Yaskawa INFORM job: A_ROOF_SIDE_0617_2_PAINT_40.JBI

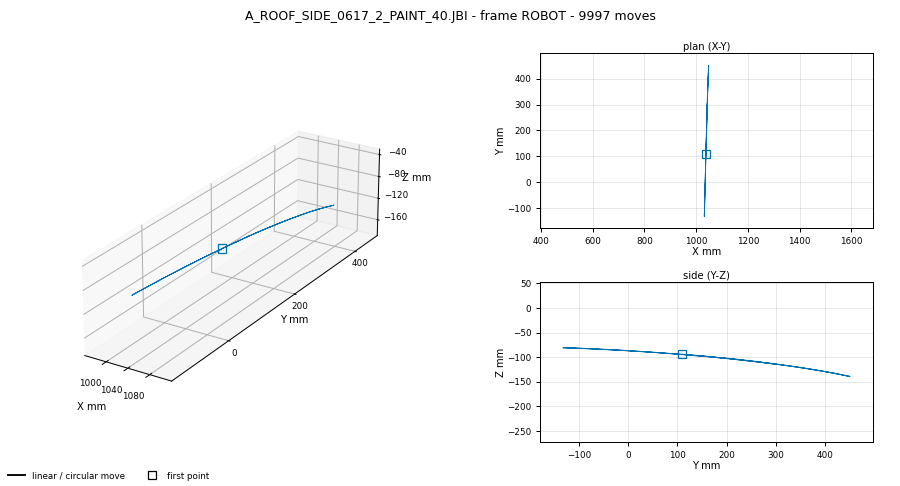
[picture p0: tool path of A_ROOF_SIDE_0617_2_PAINT_40.JBI in frame ROBOT, 9997 of 9997 moves have a stored position in this frame; points joined in program order, loops and branches not executed]
/JOB
//NAME A_ROOF_SIDE_0617_2_PAINT40
//POS
///NPOS 9997,0,0,0,0,0
///TOOL 1
///USER 0
///POSTYPE ROBOT
///RECTAN
///RCONF 1,0,0,0,0,0,0,0,0,0,0,0,0,0,0,0,0,0,0,0,0,0,0,0
C00000=1038.273,110.005,-93.623,169.688,40.047,157.538
C00001=1038.279,110.254,-93.643,169.691,40.048,157.539
C00002=1038.285,110.504,-93.663,169.693,40.048,157.539
C00003=1038.291,110.753,-93.683,169.696,40.048,157.539
C00004=1038.297,111.002,-93.703,169.698,40.048,157.539
C00005=1038.304,111.251,-93.723,169.700,40.048,157.539
C00006=1038.310,111.500,-93.743,169.702,40.049,157.539
C00007=1038.316,111.749,-93.762,169.704,40.049,157.539
C00008=1038.323,111.998,-93.782,169.706,40.049,157.539
C00009=1038.329,112.248,-93.802,169.708,40.050,157.540
C00010=1038.335,112.497,-93.822,169.710,40.049,157.540
C00011=1038.341,112.746,-93.842,169.713,40.050,157.540
C00012=1038.347,112.995,-93.862,169.715,40.050,157.540
C00013=1038.354,113.244,-93.882,169.717,40.050,157.540
C00014=1038.359,113.494,-93.903,169.719,40.051,157.540
C00015=1038.365,113.742,-93.923,169.721,40.051,157.540
C00016=1038.372,113.992,-93.943,169.723,40.051,157.540
C00017=1038.378,114.241,-93.963,169.725,40.051,157.541
C00018=1038.383,114.490,-93.984,169.727,40.052,157.541
C00019=1038.390,114.739,-94.004,169.730,40.052,157.541
C00020=1038.396,114.988,-94.024,169.732,40.052,157.541
C00021=1038.402,115.237,-94.044,169.734,40.052,157.541
C00022=1038.407,115.487,-94.065,169.736,40.053,157.541
C00023=1038.414,115.735,-94.085,169.738,40.053,157.542
C00024=1038.420,115.984,-94.105,169.740,40.053,157.542
C00025=1038.426,116.233,-94.126,169.742,40.054,157.542
C00026=1038.432,116.482,-94.146,169.745,40.054,157.542
C00027=1038.438,116.732,-94.167,169.747,40.054,157.542
C00028=1038.444,116.981,-94.187,169.749,40.054,157.542
C00029=1038.450,117.230,-94.207,169.751,40.055,157.542
C00030=1038.456,117.479,-94.227,169.753,40.055,157.543
C00031=1038.462,117.728,-94.247,169.755,40.056,157.543
C00032=1038.469,117.977,-94.268,169.757,40.055,157.543
C00033=1038.474,118.226,-94.289,169.759,40.056,157.543
C00034=1038.480,118.475,-94.309,169.762,40.056,157.543
C00035=1038.487,118.725,-94.329,169.765,40.057,157.543
C00036=1038.493,118.973,-94.349,169.767,40.057,157.543
C00037=1038.499,119.223,-94.370,169.769,40.057,157.544
C00038=1038.505,119.471,-94.391,169.771,40.057,157.544
C00039=1038.511,119.721,-94.411,169.773,40.058,157.544
C00040=1038.517,119.970,-94.431,169.775,40.058,157.544
C00041=1038.523,120.219,-94.452,169.777,40.058,157.544
C00042=1038.529,120.468,-94.472,169.780,40.059,157.544
C00043=1038.536,120.716,-94.493,169.782,40.059,157.544
C00044=1038.541,120.966,-94.514,169.784,40.059,157.544
C00045=1038.547,121.215,-94.534,169.786,40.059,157.545
C00046=1038.554,121.465,-94.554,169.788,40.060,157.545
C00047=1038.560,121.713,-94.575,169.790,40.060,157.545
C00048=1038.566,121.963,-94.596,169.792,40.060,157.545
C00049=1038.572,122.211,-94.615,169.794,40.060,157.545
C00050=1038.579,122.460,-94.637,169.797,40.061,157.545
C00051=1038.584,122.710,-94.657,169.800,40.061,157.545
C00052=1038.591,122.959,-94.677,169.802,40.061,157.546
C00053=1038.597,123.208,-94.697,169.804,40.062,157.546
C00054=1038.603,123.457,-94.719,169.806,40.061,157.546
C00055=1038.609,123.706,-94.739,169.808,40.062,157.546
C00056=1038.616,123.955,-94.759,169.810,40.062,157.546
C00057=1038.621,124.204,-94.781,169.812,40.063,157.546
C00058=1038.628,124.453,-94.801,169.814,40.062,157.546
C00059=1038.635,124.739,-94.825,169.818,40.063,157.547
C00060=1038.642,125.025,-94.849,169.820,40.063,157.547
C00061=1038.649,125.311,-94.871,169.822,40.064,157.547
C00062=1038.656,125.596,-94.895,169.825,40.064,157.547
C00063=1038.663,125.845,-94.916,169.827,40.064,157.547
C00064=1038.668,126.094,-94.937,169.829,40.064,157.547
C00065=1038.675,126.344,-94.957,169.831,40.065,157.548
C00066=1038.682,126.593,-94.978,169.833,40.065,157.548
C00067=1038.687,126.842,-94.999,169.836,40.065,157.548
C00068=1038.694,127.091,-95.020,169.838,40.065,157.548
C00069=1038.700,127.340,-95.040,169.840,40.065,157.548
C00070=1038.706,127.589,-95.061,169.843,40.066,157.548
C00071=1038.713,127.838,-95.082,169.845,40.066,157.548
C00072=1038.719,128.086,-95.102,169.847,40.067,157.549
C00073=1038.725,128.336,-95.123,169.849,40.066,157.549
C00074=1038.731,128.585,-95.143,169.851,40.067,157.549
C00075=1038.738,128.834,-95.164,169.854,40.067,157.549
C00076=1038.744,129.084,-95.185,169.856,40.067,157.549
C00077=1038.750,129.332,-95.206,169.858,40.068,157.549
C00078=1038.757,129.582,-95.226,169.861,40.068,157.549
C00079=1038.763,129.831,-95.248,169.863,40.068,157.549
C00080=1038.769,130.080,-95.268,169.865,40.068,157.550
C00081=1038.776,130.328,-95.289,169.867,40.069,157.550
C00082=1038.782,130.578,-95.310,169.869,40.068,157.550
C00083=1038.788,130.826,-95.330,169.872,40.069,157.550
C00084=1038.795,131.075,-95.351,169.874,40.069,157.550
C00085=1038.801,131.325,-95.372,169.877,40.070,157.550
C00086=1038.806,131.574,-95.394,169.879,40.070,157.551
C00087=1038.813,131.823,-95.415,169.881,40.070,157.551
C00088=1038.818,132.072,-95.435,169.883,40.070,157.551
C00089=1038.824,132.321,-95.457,169.885,40.071,157.551
C00090=1038.831,132.570,-95.478,169.888,40.071,157.551
C00091=1038.837,132.819,-95.498,169.890,40.072,157.551
C00092=1038.843,133.068,-95.520,169.892,40.072,157.551
C00093=1038.850,133.317,-95.541,169.894,40.073,157.552
C00094=1038.855,133.566,-95.562,169.896,40.072,157.552
C00095=1038.861,133.815,-95.583,169.899,40.073,157.552
C00096=1038.868,134.064,-95.604,169.901,40.073,157.552
C00097=1038.874,134.313,-95.626,169.904,40.074,157.552
C00098=1038.879,134.563,-95.646,169.906,40.074,157.552
C00099=1038.886,134.811,-95.668,169.908,40.075,157.553
C00100=1038.892,135.060,-95.689,169.910,40.074,157.553
C00101=1038.898,135.309,-95.710,169.912,40.075,157.553
C00102=1038.905,135.559,-95.731,169.914,40.075,157.553
C00103=1038.910,135.807,-95.752,169.917,40.076,157.553
C00104=1038.916,136.056,-95.774,169.920,40.076,157.553
C00105=1038.923,136.305,-95.795,169.922,40.076,157.554
C00106=1038.928,136.554,-95.815,169.924,40.076,157.554
C00107=1038.935,136.804,-95.837,169.926,40.077,157.554
C00108=1038.942,137.053,-95.858,169.928,40.077,157.554
C00109=1038.948,137.302,-95.880,169.930,40.078,157.554
C00110=1038.953,137.550,-95.901,169.933,40.078,157.554
C00111=1038.959,137.799,-95.922,169.936,40.078,157.554
C00112=1038.966,138.048,-95.944,169.938,40.079,157.555
C00113=1038.972,138.297,-95.964,169.940,40.079,157.555
C00114=1038.978,138.547,-95.986,169.942,40.079,157.555
C00115=1038.984,138.796,-96.007,169.944,40.080,157.555
C00116=1038.991,139.045,-96.028,169.947,40.080,157.555
C00117=1038.996,139.293,-96.050,169.949,40.080,157.555
C00118=1039.003,139.542,-96.071,169.952,40.081,157.556
C00119=1039.009,139.792,-96.093,169.954,40.081,157.556
C00120=1039.015,140.041,-96.115,169.956,40.082,157.556
C00121=1039.020,140.289,-96.136,169.958,40.082,157.556
C00122=1039.027,140.539,-96.157,169.960,40.083,157.556
C00123=1039.035,140.824,-96.182,169.963,40.083,157.556
C00124=1039.041,141.110,-96.206,169.966,40.083,157.557
C00125=1039.048,141.396,-96.232,169.969,40.084,157.557
C00126=1039.055,141.681,-96.255,169.971,40.084,157.557
C00127=1039.061,141.930,-96.277,169.973,40.085,157.557
C00128=1039.067,142.179,-96.299,169.976,40.085,157.557
C00129=1039.073,142.428,-96.320,169.978,40.085,157.558
C00130=1039.079,142.676,-96.342,169.981,40.086,157.558
C00131=1039.085,142.926,-96.364,169.983,40.086,157.558
C00132=1039.092,143.175,-96.386,169.985,40.087,157.558
C00133=1039.098,143.424,-96.407,169.987,40.087,157.558
C00134=1039.103,143.673,-96.429,169.990,40.088,157.558
C00135=1039.110,143.922,-96.450,169.992,40.088,157.559
C00136=1039.116,144.171,-96.472,169.995,40.088,157.559
C00137=1039.122,144.420,-96.493,169.997,40.089,157.559
C00138=1039.129,144.669,-96.514,169.999,40.089,157.559
C00139=1039.135,144.918,-96.536,170.001,40.089,157.559
C00140=1039.141,145.166,-96.558,170.004,40.089,157.559
C00141=1039.147,145.415,-96.580,170.006,40.090,157.560
C00142=1039.153,145.665,-96.601,170.008,40.090,157.560
C00143=1039.159,145.914,-96.623,170.011,40.091,157.560
C00144=1039.165,146.163,-96.645,170.013,40.091,157.560
C00145=1039.172,146.412,-96.667,170.016,40.092,157.560
C00146=1039.178,146.661,-96.689,170.018,40.092,157.560
C00147=1039.184,146.909,-96.710,170.020,40.092,157.561
C00148=1039.190,147.159,-96.732,170.022,40.093,157.561
C00149=1039.196,147.408,-96.753,170.025,40.093,157.561
C00150=1039.202,147.656,-96.775,170.028,40.094,157.561
C00151=1039.209,147.906,-96.797,170.030,40.094,157.561
C00152=1039.215,148.155,-96.819,170.032,40.095,157.562
C00153=1039.220,148.404,-96.842,170.034,40.095,157.562
C00154=1039.226,148.652,-96.863,170.036,40.095,157.562
C00155=1039.232,148.901,-96.885,170.040,40.096,157.562
C00156=1039.238,149.151,-96.906,170.042,40.096,157.562
C00157=1039.245,149.399,-96.929,170.044,40.097,157.562
C00158=1039.251,149.648,-96.950,170.046,40.097,157.563
C00159=1039.257,149.898,-96.972,170.048,40.098,157.563
C00160=1039.263,150.146,-96.995,170.051,40.098,157.563
C00161=1039.269,150.396,-97.016,170.054,40.099,157.563
C00162=1039.276,150.644,-97.039,170.056,40.099,157.563
C00163=1039.282,150.893,-97.060,170.058,40.100,157.564
C00164=1039.287,151.142,-97.082,170.060,40.100,157.564
C00165=1039.293,151.391,-97.105,170.063,40.101,157.564
C00166=1039.299,151.640,-97.126,170.066,40.101,157.564
C00167=1039.306,151.889,-97.149,170.068,40.102,157.564
C00168=1039.312,152.138,-97.170,170.070,40.102,157.565
C00169=1039.318,152.386,-97.193,170.073,40.102,157.565
C00170=1039.324,152.636,-97.215,170.075,40.103,157.565
C00171=1039.330,152.885,-97.237,170.077,40.103,157.565
C00172=1039.336,153.134,-97.259,170.079,40.104,157.565
C00173=1039.343,153.382,-97.281,170.083,40.104,157.565
C00174=1039.349,153.632,-97.303,170.085,40.104,157.566
C00175=1039.355,153.880,-97.326,170.087,40.105,157.566
C00176=1039.361,154.130,-97.347,170.089,40.106,157.566
C00177=1039.367,154.378,-97.370,170.091,40.106,157.566
C00178=1039.373,154.627,-97.391,170.095,40.107,157.567
C00179=1039.379,154.876,-97.414,170.097,40.107,157.567
C00180=1039.385,155.126,-97.436,170.099,40.108,157.567
C00181=1039.391,155.374,-97.459,170.101,40.108,157.567
C00182=1039.397,155.624,-97.481,170.104,40.108,157.567
C00183=1039.404,155.872,-97.503,170.107,40.109,157.568
C00184=1039.409,156.121,-97.526,170.109,40.110,157.568
C00185=1039.416,156.370,-97.547,170.111,40.110,157.568
C00186=1039.422,156.619,-97.570,170.114,40.111,157.568
C00187=1039.429,156.904,-97.595,170.116,40.111,157.568
C00188=1039.435,157.189,-97.621,170.120,40.112,157.569
C00189=1039.442,157.475,-97.646,170.122,40.113,157.569
C00190=1039.449,157.760,-97.672,170.125,40.113,157.569
C00191=1039.456,158.009,-97.694,170.127,40.113,157.569
C00192=1039.462,158.257,-97.716,170.130,40.114,157.569
C00193=1039.468,158.506,-97.739,170.133,40.115,157.570
C00194=1039.474,158.755,-97.762,170.135,40.115,157.570
C00195=1039.480,159.004,-97.784,170.137,40.116,157.570
C00196=1039.486,159.253,-97.806,170.140,40.116,157.570
C00197=1039.493,159.502,-97.829,170.142,40.116,157.570
C00198=1039.498,159.751,-97.852,170.144,40.117,157.571
C00199=1039.505,160.000,-97.874,170.147,40.118,157.571
C00200=1039.511,160.249,-97.897,170.150,40.118,157.571
C00201=1039.517,160.498,-97.919,170.152,40.119,157.571
C00202=1039.523,160.747,-97.942,170.154,40.120,157.572
C00203=1039.529,160.996,-97.965,170.157,40.120,157.572
C00204=1039.535,161.245,-97.988,170.160,40.121,157.572
C00205=1039.540,161.494,-98.010,170.162,40.122,157.572
C00206=1039.546,161.743,-98.032,170.164,40.122,157.572
C00207=1039.552,161.992,-98.055,170.166,40.122,157.573
C00208=1039.558,162.241,-98.078,170.170,40.123,157.573
C00209=1039.564,162.489,-98.101,170.172,40.124,157.573
C00210=1039.570,162.738,-98.124,170.174,40.124,157.573
C00211=1039.576,162.987,-98.146,170.176,40.125,157.574
C00212=1039.582,163.236,-98.169,170.179,40.126,157.574
C00213=1039.587,163.485,-98.192,170.182,40.127,157.574
C00214=1039.593,163.734,-98.215,170.184,40.127,157.574
C00215=1039.599,163.982,-98.238,170.187,40.128,157.574
C00216=1039.605,164.231,-98.261,170.189,40.129,157.575
C00217=1039.611,164.480,-98.284,170.192,40.129,157.575
C00218=1039.617,164.729,-98.306,170.194,40.130,157.575
C00219=1039.623,164.978,-98.330,170.197,40.131,157.575
C00220=1039.629,165.227,-98.352,170.199,40.131,157.576
C00221=1039.635,165.476,-98.375,170.202,40.132,157.576
C00222=1039.641,165.725,-98.398,170.204,40.132,157.576
C00223=1039.647,165.974,-98.421,170.207,40.133,157.576
C00224=1039.652,166.223,-98.444,170.209,40.134,157.577
C00225=1039.659,166.471,-98.467,170.211,40.134,157.577
C00226=1039.665,166.719,-98.490,170.215,40.135,157.577
C00227=1039.671,166.969,-98.513,170.217,40.136,157.577
C00228=1039.677,167.218,-98.536,170.219,40.136,157.577
C00229=1039.683,167.467,-98.559,170.222,40.137,157.578
C00230=1039.689,167.715,-98.582,170.224,40.138,157.578
C00231=1039.695,167.964,-98.604,170.227,40.139,157.578
C00232=1039.701,168.213,-98.627,170.230,40.139,157.579
C00233=1039.707,168.462,-98.651,170.232,40.139,157.579
C00234=1039.713,168.711,-98.674,170.234,40.140,157.579
C00235=1039.719,168.960,-98.697,170.238,40.141,157.579
C00236=1039.725,169.209,-98.720,170.240,40.142,157.579
C00237=1039.731,169.458,-98.743,170.242,40.142,157.580
C00238=1039.737,169.706,-98.766,170.245,40.143,157.580
C00239=1039.743,169.955,-98.790,170.248,40.144,157.580
C00240=1039.749,170.204,-98.813,170.250,40.144,157.580
C00241=1039.756,170.453,-98.835,170.253,40.145,157.581
C00242=1039.761,170.702,-98.858,170.255,40.146,157.581
C00243=1039.768,170.951,-98.882,170.257,40.146,157.581
C00244=1039.774,171.200,-98.905,170.261,40.147,157.581
C00245=1039.779,171.449,-98.928,170.263,40.147,157.582
C00246=1039.785,171.697,-98.951,170.265,40.148,157.582
C00247=1039.792,171.946,-98.975,170.268,40.149,157.582
C00248=1039.798,172.195,-98.997,170.271,40.149,157.582
C00249=1039.804,172.444,-99.020,170.273,40.150,157.583
C00250=1039.810,172.692,-99.044,170.276,40.151,157.583
C00251=1039.817,172.978,-99.070,170.279,40.152,157.583
C00252=1039.824,173.262,-99.097,170.282,40.152,157.583
C00253=1039.831,173.547,-99.123,170.285,40.153,157.584
C00254=1039.838,173.831,-99.150,170.288,40.154,157.584
C00255=1039.844,174.080,-99.173,170.290,40.154,157.584
C00256=1039.850,174.330,-99.196,170.294,40.155,157.584
C00257=1039.857,174.578,-99.220,170.296,40.156,157.585
C00258=1039.862,174.827,-99.243,170.298,40.156,157.585
C00259=1039.869,175.076,-99.267,170.301,40.157,157.585
C00260=1039.875,175.325,-99.289,170.303,40.158,157.585
C00261=1039.881,175.574,-99.312,170.307,40.159,157.586
C00262=1039.888,175.823,-99.336,170.309,40.159,157.586
C00263=1039.893,176.071,-99.359,170.311,40.160,157.586
C00264=1039.899,176.320,-99.383,170.314,40.160,157.586
C00265=1039.906,176.569,-99.406,170.317,40.161,157.587
C00266=1039.912,176.818,-99.430,170.320,40.162,157.587
C00267=1039.918,177.067,-99.453,170.322,40.162,157.587
C00268=1039.925,177.315,-99.476,170.324,40.163,157.587
C00269=1039.931,177.564,-99.499,170.328,40.164,157.587
C00270=1039.937,177.813,-99.523,170.330,40.165,157.588
C00271=1039.943,178.062,-99.546,170.333,40.165,157.588
C00272=1039.949,178.310,-99.570,170.335,40.166,157.588
C00273=1039.955,178.560,-99.593,170.339,40.166,157.589
C00274=1039.961,178.808,-99.617,170.341,40.168,157.589
C00275=1039.968,179.058,-99.640,170.344,40.168,157.589
C00276=1039.974,179.306,-99.664,170.346,40.169,157.589
C00277=1039.981,179.555,-99.687,170.350,40.169,157.590
C00278=1039.987,179.804,-99.710,170.352,40.170,157.590
C00279=1039.994,180.053,-99.734,170.354,40.171,157.590
C00280=1039.999,180.301,-99.757,170.357,40.171,157.590
C00281=1040.005,180.550,-99.781,170.359,40.172,157.591
C00282=1040.012,180.799,-99.805,170.363,40.172,157.591
C00283=1040.018,181.048,-99.828,170.365,40.174,157.591
C00284=1040.024,181.297,-99.852,170.368,40.174,157.591
C00285=1040.030,181.545,-99.876,170.370,40.175,157.592
C00286=1040.037,181.794,-99.899,170.374,40.175,157.592
C00287=1040.044,182.042,-99.922,170.376,40.176,157.592
C00288=1040.050,182.291,-99.946,170.379,40.177,157.592
C00289=1040.056,182.540,-99.969,170.381,40.178,157.593
C00290=1040.063,182.789,-99.993,170.385,40.178,157.593
C00291=1040.069,183.038,-100.017,170.387,40.179,157.593
C00292=1040.075,183.287,-100.041,170.390,40.179,157.593
C00293=1040.082,183.536,-100.064,170.392,40.180,157.594
C00294=1040.087,183.785,-100.088,170.396,40.181,157.594
C00295=1040.093,184.034,-100.112,170.398,40.182,157.594
C00296=1040.099,184.282,-100.136,170.401,40.183,157.594
C00297=1040.105,184.531,-100.160,170.404,40.184,157.595
C00298=1040.111,184.780,-100.184,170.406,40.185,157.595
C00299=1040.117,185.028,-100.208,170.409,40.186,157.595
C00300=1040.123,185.277,-100.232,170.411,40.186,157.596
C00301=1040.129,185.526,-100.257,170.415,40.187,157.596
C00302=1040.135,185.775,-100.281,170.417,40.188,157.596
C00303=1040.141,186.023,-100.305,170.420,40.189,157.597
C00304=1040.147,186.272,-100.329,170.423,40.190,157.597
C00305=1040.153,186.521,-100.353,170.426,40.191,157.597
C00306=1040.159,186.770,-100.377,170.428,40.192,157.597
C00307=1040.164,187.018,-100.402,170.431,40.193,157.598
C00308=1040.171,187.267,-100.426,170.434,40.194,157.598
C00309=1040.176,187.516,-100.450,170.437,40.195,157.598
C00310=1040.183,187.765,-100.474,170.439,40.196,157.599
C00311=1040.188,188.014,-100.498,170.443,40.196,157.599
C00312=1040.195,188.262,-100.522,170.445,40.197,157.599
C00313=1040.200,188.511,-100.546,170.448,40.198,157.599
C00314=1040.207,188.760,-100.570,170.450,40.199,157.600
C00315=1040.214,189.044,-100.598,170.454,40.200,157.600
C00316=1040.221,189.328,-100.625,170.457,40.201,157.600
C00317=1040.227,189.613,-100.654,170.460,40.202,157.601
C00318=1040.234,189.897,-100.681,170.463,40.203,157.601
C00319=1040.240,190.146,-100.705,170.466,40.204,157.601
C00320=1040.247,190.395,-100.730,170.469,40.205,157.602
C00321=1040.253,190.643,-100.754,170.472,40.206,157.602
C00322=1040.259,190.892,-100.779,170.475,40.207,157.602
C00323=1040.265,191.141,-100.802,170.477,40.208,157.603
C00324=1040.271,191.390,-100.827,170.481,40.209,157.603
C00325=1040.277,191.638,-100.852,170.483,40.209,157.603
C00326=1040.283,191.887,-100.876,170.486,40.210,157.604
C00327=1040.289,192.136,-100.900,170.488,40.211,157.604
C00328=1040.295,192.385,-100.925,170.492,40.212,157.604
C00329=1040.302,192.633,-100.949,170.494,40.213,157.605
C00330=1040.308,192.882,-100.974,170.497,40.214,157.605
C00331=1040.313,193.131,-100.998,170.500,40.215,157.605
C00332=1040.319,193.380,-101.022,170.503,40.216,157.606
C00333=1040.326,193.628,-101.047,170.506,40.217,157.606
C00334=1040.332,193.877,-101.071,170.509,40.218,157.606
C00335=1040.338,194.126,-101.096,170.512,40.219,157.606
C00336=1040.345,194.374,-101.120,170.514,40.220,157.607
C00337=1040.350,194.623,-101.145,170.518,40.221,157.607
C00338=1040.357,194.872,-101.169,170.520,40.222,157.607
C00339=1040.363,195.120,-101.194,170.523,40.223,157.608
C00340=1040.369,195.369,-101.218,170.527,40.224,157.608
C00341=1040.375,195.617,-101.243,170.529,40.225,157.608
C00342=1040.381,195.867,-101.268,170.532,40.226,157.609
C00343=1040.387,196.116,-101.292,170.534,40.227,157.609
C00344=1040.394,196.364,-101.317,170.538,40.228,157.609
C00345=1040.400,196.613,-101.341,170.541,40.229,157.610
C00346=1040.406,196.861,-101.366,170.543,40.230,157.610
C00347=1040.413,197.110,-101.390,170.547,40.231,157.610
C00348=1040.419,197.359,-101.415,170.549,40.232,157.611
C00349=1040.425,197.608,-101.439,170.552,40.233,157.611
C00350=1040.431,197.856,-101.464,170.556,40.233,157.611
C00351=1040.437,198.105,-101.489,170.558,40.234,157.611
C00352=1040.444,198.353,-101.514,170.561,40.235,157.612
C00353=1040.450,198.603,-101.538,170.565,40.236,157.612
C00354=1040.457,198.851,-101.563,170.567,40.237,157.612
C00355=1040.462,199.100,-101.587,170.570,40.238,157.613
C00356=1040.469,199.348,-101.612,170.572,40.239,157.613
C00357=1040.475,199.597,-101.637,170.576,40.240,157.613
C00358=1040.481,199.846,-101.662,170.579,40.241,157.614
C00359=1040.488,200.095,-101.686,170.581,40.242,157.614
C00360=1040.494,200.344,-101.711,170.585,40.243,157.614
C00361=1040.500,200.591,-101.736,170.588,40.244,157.615
C00362=1040.506,200.841,-101.760,170.590,40.245,157.615
C00363=1040.512,201.089,-101.786,170.594,40.246,157.615
C00364=1040.519,201.338,-101.811,170.597,40.247,157.616
C00365=1040.525,201.587,-101.835,170.600,40.248,157.616
C00366=1040.531,201.836,-101.860,170.603,40.249,157.616
C00367=1040.537,202.084,-101.885,170.606,40.250,157.617
C00368=1040.543,202.333,-101.910,170.609,40.251,157.617
C00369=1040.549,202.582,-101.935,170.612,40.253,157.618
C00370=1040.555,202.830,-101.961,170.614,40.254,157.618
C00371=1040.562,203.079,-101.986,170.618,40.255,157.618
C00372=1040.568,203.328,-102.011,170.621,40.256,157.619
C00373=1040.574,203.577,-102.036,170.623,40.257,157.619
C00374=1040.579,203.825,-102.061,170.627,40.259,157.619
C00375=1040.585,204.073,-102.086,170.630,40.259,157.620
C00376=1040.592,204.322,-102.112,170.632,40.261,157.620
C00377=1040.599,204.571,-102.136,170.636,40.261,157.620
C00378=1040.605,204.819,-102.162,170.639,40.263,157.621
C00379=1040.631,205.871,-102.268,170.925,40.366,157.654
C00380=1040.639,206.173,-102.300,170.927,40.368,157.655
C00381=1040.647,206.477,-102.333,170.930,40.370,157.656
C00382=1040.655,206.780,-102.365,170.933,40.373,157.656
C00383=1040.664,207.084,-102.396,170.935,40.375,157.657
C00384=1040.670,207.333,-102.423,170.938,40.377,157.657
C00385=1040.677,207.581,-102.449,170.939,40.379,157.658
C00386=1040.684,207.830,-102.476,170.942,40.380,157.658
C00387=1040.689,208.078,-102.502,170.944,40.383,157.659
C00388=1040.697,208.326,-102.530,170.946,40.384,157.659
C00389=1040.703,208.574,-102.556,170.948,40.386,157.660
C00390=1040.710,208.823,-102.583,170.951,40.388,157.660
C00391=1040.717,209.072,-102.609,170.952,40.390,157.661
C00392=1040.723,209.320,-102.635,170.955,40.392,157.661
C00393=1040.730,209.569,-102.662,170.957,40.393,157.662
C00394=1040.736,209.817,-102.688,170.959,40.396,157.662
C00395=1040.743,210.066,-102.715,170.962,40.397,157.663
C00396=1040.750,210.315,-102.742,170.964,40.399,157.663
C00397=1040.757,210.562,-102.768,170.967,40.401,157.664
C00398=1040.764,210.811,-102.795,170.968,40.403,157.664
C00399=1040.769,211.059,-102.821,170.971,40.405,157.665
C00400=1040.777,211.308,-102.848,170.973,40.407,157.665
C00401=1040.783,211.557,-102.875,170.976,40.409,157.666
C00402=1040.790,211.805,-102.902,170.977,40.410,157.666
C00403=1040.796,212.054,-102.929,170.980,40.413,157.667
C00404=1040.803,212.302,-102.955,170.982,40.414,157.667
C00405=1040.809,212.551,-102.982,170.984,40.416,157.668
C00406=1040.816,212.799,-103.009,170.986,40.418,157.668
C00407=1040.822,213.047,-103.035,170.989,40.420,157.669
C00408=1040.829,213.296,-103.062,170.991,40.422,157.669
C00409=1040.836,213.544,-103.090,170.993,40.424,157.670
C00410=1040.843,213.792,-103.116,170.995,40.426,157.670
C00411=1040.849,214.042,-103.143,170.998,40.428,157.671
C00412=1040.856,214.290,-103.170,171.001,40.430,157.671
C00413=1040.862,214.538,-103.196,171.002,40.431,157.672
C00414=1040.868,214.787,-103.223,171.005,40.434,157.672
C00415=1040.876,215.035,-103.251,171.007,40.435,157.673
C00416=1040.882,215.284,-103.277,171.010,40.437,157.673
C00417=1040.889,215.532,-103.304,171.012,40.439,157.674
C00418=1040.895,215.781,-103.331,171.014,40.441,157.674
C00419=1040.903,216.030,-103.358,171.016,40.443,157.675
C00420=1040.909,216.277,-103.385,171.019,40.444,157.675
C00421=1040.915,216.526,-103.412,171.021,40.446,157.676
C00422=1040.922,216.775,-103.439,171.023,40.448,157.676
C00423=1040.928,217.023,-103.466,171.025,40.450,157.676
C00424=1040.935,217.272,-103.492,171.028,40.452,157.677
C00425=1040.942,217.520,-103.520,171.030,40.454,157.678
C00426=1040.949,217.769,-103.547,171.033,40.455,157.678
C00427=1040.955,218.017,-103.574,171.035,40.458,157.679
C00428=1040.962,218.266,-103.601,171.037,40.459,157.679
C00429=1040.969,218.514,-103.628,171.040,40.461,157.679
C00430=1040.975,218.763,-103.655,171.042,40.463,157.680
C00431=1040.982,219.010,-103.682,171.045,40.465,157.681
C00432=1040.989,219.259,-103.709,171.047,40.467,157.681
C00433=1040.996,219.507,-103.736,171.049,40.468,157.681
C00434=1041.002,219.756,-103.763,171.051,40.471,157.682
C00435=1041.009,220.005,-103.791,171.054,40.472,157.682
C00436=1041.018,220.313,-103.824,171.056,40.474,157.683
C00437=1041.025,220.622,-103.858,171.060,40.477,157.684
C00438=1041.033,220.931,-103.892,171.063,40.479,157.684
C00439=1041.042,221.240,-103.926,171.065,40.482,157.685
C00440=1041.049,221.488,-103.954,171.068,40.483,157.685
C00441=1041.055,221.737,-103.981,171.071,40.486,157.686
C00442=1041.061,221.985,-104.008,171.073,40.487,157.687
C00443=1041.068,222.233,-104.036,171.076,40.489,157.687
C00444=1041.075,222.482,-104.062,171.077,40.491,157.688
C00445=1041.081,222.730,-104.090,171.080,40.493,157.688
C00446=1041.088,222.979,-104.118,171.082,40.495,157.688
C00447=1041.094,223.227,-104.145,171.085,40.497,157.689
C00448=1041.101,223.476,-104.172,171.087,40.498,157.690
C00449=1041.107,223.724,-104.200,171.090,40.500,157.690
C00450=1041.114,223.973,-104.227,171.092,40.502,157.691
C00451=1041.121,224.221,-104.255,171.094,40.504,157.691
C00452=1041.128,224.470,-104.282,171.097,40.506,157.692
C00453=1041.134,224.718,-104.309,171.099,40.508,157.692
C00454=1041.141,224.966,-104.337,171.101,40.510,157.693
C00455=1041.147,225.214,-104.364,171.104,40.512,157.693
C00456=1041.154,225.463,-104.392,171.107,40.513,157.694
C00457=1041.161,225.711,-104.420,171.109,40.515,157.694
C00458=1041.168,225.960,-104.446,171.112,40.517,157.695
C00459=1041.174,226.209,-104.474,171.114,40.519,157.695
C00460=1041.180,226.456,-104.501,171.116,40.521,157.696
C00461=1041.187,226.705,-104.529,171.118,40.523,157.696
C00462=1041.194,226.953,-104.557,171.121,40.525,157.697
C00463=1041.200,227.202,-104.585,171.123,40.526,157.697
C00464=1041.207,227.450,-104.612,171.126,40.529,157.698
C00465=1041.214,227.698,-104.640,171.128,40.530,157.698
C00466=1041.221,227.947,-104.668,171.131,40.532,157.699
C00467=1041.228,228.196,-104.694,171.134,40.534,157.699
C00468=1041.234,228.444,-104.722,171.136,40.536,157.700
C00469=1041.241,228.693,-104.750,171.139,40.537,157.700
C00470=1041.248,228.941,-104.777,171.141,40.540,157.701
C00471=1041.254,229.190,-104.806,171.144,40.541,157.701
C00472=1041.260,229.437,-104.834,171.146,40.543,157.702
C00473=1041.267,229.685,-104.862,171.149,40.545,157.702
C00474=1041.273,229.934,-104.889,171.150,40.547,157.703
C00475=1041.280,230.182,-104.917,171.153,40.549,157.703
C00476=1041.287,230.431,-104.945,171.155,40.551,157.704
C00477=1041.293,230.679,-104.972,171.158,40.553,157.704
C00478=1041.300,230.927,-105.000,171.161,40.555,157.705
C00479=1041.307,231.176,-105.028,171.163,40.556,157.705
C00480=1041.313,231.424,-105.056,171.166,40.558,157.706
C00481=1041.319,231.673,-105.084,171.168,40.560,157.706
C00482=1041.326,231.921,-105.112,171.171,40.562,157.707
C00483=1041.333,232.169,-105.140,171.173,40.564,157.707
C00484=1041.340,232.418,-105.168,171.176,40.566,157.708
C00485=1041.346,232.666,-105.196,171.179,40.568,157.708
C00486=1041.352,232.915,-105.224,171.181,40.569,157.709
C00487=1041.359,233.163,-105.252,171.184,40.572,157.709
C00488=1041.366,233.411,-105.280,171.186,40.573,157.710
C00489=1041.373,233.660,-105.308,171.189,40.576,157.710
C00490=1041.379,233.908,-105.336,171.191,40.577,157.711
C00491=1041.386,234.156,-105.365,171.194,40.579,157.712
C00492=1041.393,234.457,-105.398,171.197,40.582,157.712
C00493=1041.401,234.759,-105.432,171.200,40.584,157.713
C00494=1041.410,235.060,-105.466,171.203,40.586,157.713
C00495=1041.418,235.362,-105.501,171.206,40.588,157.714
C00496=1041.424,235.610,-105.529,171.208,40.590,157.715
C00497=1041.431,235.858,-105.556,171.211,40.592,157.715
C00498=1041.437,236.107,-105.585,171.213,40.594,157.715
C00499=1041.444,236.355,-105.613,171.217,40.596,157.716
C00500=1041.451,236.603,-105.641,171.219,40.597,157.717
C00501=1041.457,236.852,-105.670,171.222,40.600,157.717
C00502=1041.464,237.100,-105.698,171.224,40.601,157.718
C00503=1041.471,237.348,-105.726,171.227,40.604,157.718
C00504=1041.477,237.596,-105.754,171.230,40.605,157.719
C00505=1041.483,237.845,-105.782,171.232,40.607,157.719
C00506=1041.490,238.093,-105.811,171.235,40.609,157.720
C00507=1041.497,238.342,-105.839,171.237,40.611,157.720
C00508=1041.504,238.590,-105.868,171.240,40.613,157.721
C00509=1041.510,238.839,-105.895,171.242,40.615,157.721
C00510=1041.517,239.086,-105.924,171.245,40.617,157.722
C00511=1041.523,239.335,-105.952,171.248,40.618,157.722
C00512=1041.530,239.583,-105.981,171.250,40.620,157.723
C00513=1041.537,239.831,-106.008,171.253,40.622,157.723
C00514=1041.543,240.080,-106.037,171.255,40.624,157.724
C00515=1041.550,240.328,-106.065,171.258,40.626,157.724
C00516=1041.557,240.577,-106.094,171.260,40.628,157.725
C00517=1041.563,240.825,-106.122,171.263,40.630,157.726
C00518=1041.570,241.073,-106.151,171.267,40.631,157.726
C00519=1041.577,241.321,-106.180,171.269,40.634,157.727
C00520=1041.583,241.570,-106.207,171.272,40.635,157.727
C00521=1041.590,241.818,-106.237,171.274,40.638,157.728
C00522=1041.596,242.066,-106.266,171.277,40.639,157.728
C00523=1041.603,242.315,-106.294,171.279,40.641,157.729
C00524=1041.609,242.563,-106.323,171.282,40.643,157.729
C00525=1041.616,242.811,-106.351,171.285,40.645,157.730
C00526=1041.623,243.059,-106.380,171.287,40.647,157.730
C00527=1041.629,243.308,-106.408,171.290,40.649,157.731
C00528=1041.636,243.556,-106.437,171.292,40.651,157.731
C00529=1041.642,243.804,-106.466,171.295,40.653,157.732
C00530=1041.649,244.052,-106.495,171.297,40.655,157.732
C00531=1041.655,244.301,-106.523,171.301,40.657,157.733
C00532=1041.662,244.549,-106.552,171.304,40.658,157.733
C00533=1041.669,244.797,-106.581,171.306,40.660,157.734
C00534=1041.675,245.045,-106.610,171.309,40.662,157.735
C00535=1041.682,245.294,-106.638,171.311,40.664,157.735
C00536=1041.688,245.543,-106.667,171.314,40.667,157.736
C00537=1041.695,245.791,-106.696,171.317,40.668,157.736
C00538=1041.701,246.039,-106.725,171.319,40.670,157.737
C00539=1041.707,246.287,-106.754,171.322,40.672,157.737
C00540=1041.713,246.535,-106.783,171.325,40.674,157.738
C00541=1041.721,246.784,-106.812,171.328,40.676,157.739
C00542=1041.727,247.032,-106.841,171.331,40.678,157.739
C00543=1041.733,247.280,-106.870,171.333,40.680,157.740
C00544=1041.740,247.528,-106.899,171.336,40.682,157.740
C00545=1041.746,247.776,-106.928,171.338,40.684,157.741
C00546=1041.753,248.025,-106.957,171.341,40.686,157.741
C00547=1041.759,248.273,-106.986,171.344,40.688,157.742
C00548=1041.767,248.569,-107.021,171.347,40.691,157.742
C00549=1041.774,248.864,-107.055,171.351,40.693,157.743
C00550=1041.783,249.160,-107.090,171.354,40.695,157.744
C00551=1041.791,249.455,-107.125,171.358,40.698,157.744
C00552=1041.797,249.703,-107.154,171.360,40.699,157.745
C00553=1041.803,249.951,-107.183,171.363,40.701,157.746
C00554=1041.809,250.199,-107.212,171.365,40.704,157.746
C00555=1041.816,250.448,-107.241,171.368,40.705,157.747
C00556=1041.823,250.696,-107.270,171.372,40.707,157.747
C00557=1041.830,250.944,-107.299,171.374,40.709,157.748
C00558=1041.837,251.192,-107.329,171.377,40.711,157.748
C00559=1041.843,251.441,-107.358,171.379,40.713,157.749
C00560=1041.849,251.689,-107.387,171.382,40.715,157.749
C00561=1041.856,251.938,-107.416,171.386,40.717,157.750
C00562=1041.862,252.186,-107.445,171.388,40.719,157.750
C00563=1041.869,252.433,-107.475,171.391,40.721,157.751
C00564=1041.876,252.682,-107.504,171.393,40.723,157.752
C00565=1041.882,252.930,-107.534,171.396,40.725,157.752
C00566=1041.889,253.178,-107.562,171.400,40.727,157.753
C00567=1041.896,253.427,-107.591,171.402,40.729,157.753
C00568=1041.902,253.674,-107.621,171.405,40.731,157.754
C00569=1041.909,253.922,-107.650,171.407,40.733,157.754
C00570=1041.915,254.171,-107.680,171.410,40.735,157.755
C00571=1041.922,254.419,-107.709,171.414,40.737,157.756
C00572=1041.929,254.668,-107.739,171.416,40.739,157.756
C00573=1041.935,254.916,-107.768,171.419,40.741,157.757
C00574=1041.941,255.164,-107.797,171.421,40.743,157.757
C00575=1041.949,255.412,-107.827,171.425,40.744,157.758
C00576=1041.955,255.660,-107.856,171.428,40.746,157.758
C00577=1041.963,255.908,-107.886,171.430,40.749,157.759
C00578=1041.969,256.156,-107.915,171.434,40.750,157.759
C00579=1041.975,256.404,-107.944,171.436,40.752,157.760
C00580=1041.982,256.653,-107.974,171.439,40.754,157.761
C00581=1041.989,256.901,-108.003,171.442,40.756,157.761
C00582=1041.996,257.149,-108.033,171.445,40.758,157.762
C00583=1042.002,257.397,-108.062,171.448,40.760,157.762
C00584=1042.009,257.646,-108.091,171.450,40.762,157.763
C00585=1042.015,257.893,-108.121,171.454,40.764,157.763
C00586=1042.022,258.142,-108.150,171.457,40.766,157.764
C00587=1042.029,258.390,-108.180,171.459,40.768,157.765
C00588=1042.036,258.639,-108.210,171.462,40.770,157.765
C00589=1042.042,258.886,-108.239,171.465,40.772,157.766
C00590=1042.050,259.135,-108.268,171.468,40.774,157.766
C00591=1042.056,259.382,-108.298,171.471,40.776,157.767
C00592=1042.063,259.631,-108.327,171.474,40.778,157.767
C00593=1042.070,259.878,-108.357,171.477,40.779,157.768
C00594=1042.077,260.127,-108.387,171.479,40.781,157.768
C00595=1042.084,260.376,-108.417,171.483,40.784,157.769
C00596=1042.090,260.623,-108.446,171.486,40.785,157.770
C00597=1042.097,260.872,-108.476,171.488,40.787,157.770
C00598=1042.104,261.119,-108.506,171.492,40.789,157.771
C00599=1042.111,261.368,-108.535,171.495,40.791,157.771
C00600=1042.117,261.616,-108.565,171.497,40.793,157.772
C00601=1042.124,261.864,-108.595,171.501,40.795,157.772
C00602=1042.131,262.113,-108.624,171.503,40.797,157.773
C00603=1042.138,262.360,-108.654,171.507,40.799,157.774
C00604=1042.146,262.654,-108.689,171.510,40.801,157.774
C00605=1042.153,262.948,-108.726,171.514,40.804,157.775
C00606=1042.161,263.243,-108.761,171.517,40.806,157.776
C00607=1042.169,263.537,-108.796,171.521,40.809,157.776
C00608=1042.176,263.785,-108.826,171.524,40.811,157.777
C00609=1042.182,264.033,-108.857,171.526,40.812,157.777
C00610=1042.189,264.281,-108.887,171.530,40.815,157.778
C00611=1042.195,264.528,-108.916,171.533,40.817,157.779
C00612=1042.202,264.778,-108.946,171.535,40.819,157.779
C00613=1042.209,265.026,-108.977,171.539,40.821,157.780
C00614=1042.215,265.273,-109.006,171.541,40.823,157.780
C00615=1042.222,265.522,-109.037,171.545,40.825,157.781
C00616=1042.228,265.769,-109.067,171.548,40.827,157.782
C00617=1042.235,266.018,-109.097,171.551,40.829,157.782
C00618=1042.242,266.266,-109.128,171.554,40.831,157.783
C00619=1042.248,266.514,-109.157,171.557,40.833,157.783
C00620=1042.255,266.762,-109.188,171.559,40.835,157.784
C00621=1042.262,267.010,-109.218,171.563,40.837,157.785
C00622=1042.268,267.258,-109.248,171.566,40.839,157.785
C00623=1042.276,267.506,-109.278,171.569,40.841,157.786
C00624=1042.282,267.755,-109.309,171.572,40.844,157.786
C00625=1042.289,268.002,-109.339,171.575,40.845,157.787
C00626=1042.295,268.251,-109.369,171.578,40.847,157.788
C00627=1042.302,268.499,-109.399,171.581,40.849,157.788
C00628=1042.308,268.747,-109.430,171.585,40.852,157.789
C00629=1042.315,268.995,-109.460,171.587,40.854,157.789
C00630=1042.322,269.243,-109.491,171.591,40.856,157.790
C00631=1042.328,269.490,-109.521,171.594,40.858,157.791
C00632=1042.335,269.739,-109.552,171.596,40.860,157.791
C00633=1042.342,269.987,-109.582,171.600,40.862,157.792
C00634=1042.348,270.235,-109.612,171.603,40.864,157.792
C00635=1042.355,270.483,-109.642,171.606,40.866,157.793
C00636=1042.362,270.731,-109.674,171.609,40.868,157.794
C00637=1042.368,270.978,-109.704,171.613,40.870,157.794
C00638=1042.375,271.227,-109.734,171.615,40.872,157.795
C00639=1042.382,271.475,-109.764,171.619,40.875,157.796
C00640=1042.389,271.723,-109.796,171.622,40.877,157.796
C00641=1042.394,271.971,-109.826,171.624,40.879,157.797
C00642=1042.402,272.219,-109.856,171.628,40.881,157.797
C00643=1042.408,272.467,-109.888,171.631,40.883,157.798
C00644=1042.415,272.715,-109.918,171.634,40.885,157.799
C00645=1042.421,272.963,-109.948,171.637,40.887,157.799
C00646=1042.428,273.211,-109.980,171.641,40.889,157.800
C00647=1042.435,273.459,-110.010,171.643,40.891,157.800
C00648=1042.442,273.708,-110.041,171.647,40.893,157.801
C00649=1042.448,273.955,-110.072,171.650,40.895,157.802
C00650=1042.455,274.203,-110.102,171.653,40.897,157.802
C00651=1042.462,274.451,-110.133,171.656,40.900,157.803
C00652=1042.468,274.700,-110.164,171.660,40.902,157.804
C00653=1042.475,274.947,-110.195,171.662,40.904,157.804
C00654=1042.481,275.195,-110.225,171.666,40.906,157.805
C00655=1042.488,275.443,-110.256,171.669,40.908,157.805
C00656=1042.494,275.691,-110.287,171.672,40.910,157.806
C00657=1042.502,275.939,-110.318,171.675,40.912,157.807
C00658=1042.508,276.188,-110.349,171.679,40.914,157.807
C00659=1042.514,276.435,-110.380,171.682,40.917,157.808
C00660=1042.523,276.733,-110.417,171.685,40.919,157.809
C00661=1042.530,277.032,-110.454,171.689,40.922,157.809
C00662=1042.539,277.331,-110.491,171.693,40.925,157.810
C00663=1042.547,277.630,-110.529,171.697,40.927,157.811
C00664=1042.553,277.877,-110.560,171.701,40.929,157.812
C00665=1042.560,278.125,-110.590,171.704,40.931,157.812
C00666=1042.567,278.373,-110.622,171.707,40.934,157.813
C00667=1042.574,278.621,-110.653,171.711,40.936,157.814
C00668=1042.580,278.870,-110.684,171.713,40.938,157.814
C00669=1042.587,279.117,-110.715,171.717,40.940,157.815
C00670=1042.594,279.365,-110.747,171.720,40.942,157.815
C00671=1042.600,279.613,-110.778,171.724,40.945,157.816
C00672=1042.606,279.861,-110.809,171.726,40.947,157.817
C00673=1042.613,280.109,-110.840,171.730,40.949,157.817
C00674=1042.620,280.357,-110.871,171.734,40.951,157.818
C00675=1042.626,280.605,-110.903,171.736,40.953,157.819
C00676=1042.633,280.853,-110.934,171.740,40.955,157.819
C00677=1042.640,281.101,-110.965,171.743,40.958,157.820
C00678=1042.646,281.349,-110.996,171.747,40.960,157.821
C00679=1042.653,281.597,-111.028,171.749,40.962,157.821
C00680=1042.660,281.845,-111.059,171.753,40.964,157.822
C00681=1042.666,282.093,-111.091,171.757,40.967,157.823
C00682=1042.673,282.341,-111.122,171.760,40.969,157.823
C00683=1042.680,282.589,-111.154,171.763,40.971,157.824
C00684=1042.687,282.837,-111.185,171.766,40.974,157.825
C00685=1042.693,283.084,-111.216,171.770,40.976,157.825
C00686=1042.700,283.332,-111.248,171.773,40.978,157.826
C00687=1042.707,283.580,-111.279,171.776,40.980,157.827
C00688=1042.714,283.828,-111.311,171.780,40.983,157.827
C00689=1042.720,284.076,-111.342,171.783,40.985,157.828
C00690=1042.727,284.324,-111.374,171.786,40.987,157.829
C00691=1042.734,284.572,-111.405,171.790,40.989,157.829
C00692=1042.740,284.820,-111.437,171.793,40.992,157.830
C00693=1042.747,285.068,-111.468,171.797,40.994,157.831
C00694=1042.754,285.316,-111.499,171.800,40.996,157.831
C00695=1042.761,285.564,-111.531,171.803,40.998,157.832
C00696=1042.767,285.811,-111.562,171.807,41.000,157.833
C00697=1042.774,286.059,-111.594,171.811,41.003,157.833
C00698=1042.781,286.307,-111.626,171.813,41.005,157.834
C00699=1042.788,286.554,-111.657,171.817,41.007,157.835
C00700=1042.795,286.802,-111.689,171.821,41.009,157.835
C00701=1042.801,287.050,-111.720,171.824,41.012,157.836
C00702=1042.808,287.298,-111.752,171.827,41.014,157.837
C00703=1042.814,287.546,-111.784,171.831,41.016,157.837
C00704=1042.821,287.794,-111.816,171.834,41.019,157.838
C00705=1042.828,288.042,-111.848,171.837,41.021,157.839
C00706=1042.835,288.290,-111.880,171.841,41.023,157.839
C00707=1042.841,288.538,-111.912,171.844,41.025,157.840
C00708=1042.848,288.786,-111.943,171.848,41.027,157.841
C00709=1042.855,289.033,-111.975,171.851,41.029,157.841
C00710=1042.862,289.281,-112.007,171.854,41.032,157.842
C00711=1042.868,289.529,-112.039,171.858,41.034,157.843
C00712=1042.875,289.776,-112.071,171.862,41.037,157.844
C00713=1042.882,290.025,-112.103,171.866,41.039,157.844
C00714=1042.889,290.272,-112.135,171.868,41.041,157.845
C00715=1042.895,290.520,-112.167,171.872,41.044,157.846
C00716=1042.904,290.830,-112.207,171.876,41.046,157.846
C00717=1042.912,291.141,-112.247,171.881,41.050,157.847
C00718=1042.921,291.451,-112.288,171.885,41.052,157.848
C00719=1042.929,291.761,-112.327,171.890,41.055,157.849
C00720=1042.936,292.010,-112.360,171.893,41.058,157.850
C00721=1042.942,292.258,-112.391,171.897,41.060,157.851
C00722=1042.950,292.505,-112.423,171.900,41.062,157.851
C00723=1042.955,292.753,-112.455,171.904,41.065,157.852
C00724=1042.963,293.000,-112.488,171.907,41.067,157.853
C00725=1042.970,293.248,-112.520,171.911,41.070,157.853
C00726=1042.976,293.497,-112.552,171.914,41.072,157.854
C00727=1042.983,293.744,-112.584,171.918,41.074,157.855
C00728=1042.990,293.991,-112.616,171.921,41.077,157.856
C00729=1042.997,294.240,-112.649,171.925,41.079,157.856
C00730=1043.004,294.487,-112.681,171.929,41.081,157.857
C00731=1043.010,294.735,-112.714,171.933,41.084,157.858
C00732=1043.017,294.983,-112.745,171.936,41.086,157.858
C00733=1043.024,295.231,-112.778,171.939,41.089,157.859
C00734=1043.031,295.478,-112.810,171.943,41.091,157.860
C00735=1043.037,295.726,-112.843,171.947,41.093,157.861
C00736=1043.043,295.974,-112.876,171.951,41.096,157.861
C00737=1043.051,296.222,-112.908,171.953,41.098,157.862
C00738=1043.057,296.470,-112.940,171.957,41.101,157.863
C00739=1043.063,296.717,-112.973,171.961,41.103,157.864
C00740=1043.070,296.965,-113.006,171.965,41.105,157.864
C00741=1043.077,297.213,-113.038,171.969,41.108,157.865
C00742=1043.083,297.461,-113.071,171.971,41.111,157.866
C00743=1043.090,297.708,-113.104,171.975,41.113,157.867
C00744=1043.096,297.956,-113.137,171.979,41.115,157.867
C00745=1043.103,298.204,-113.170,171.983,41.118,157.868
C00746=1043.110,298.451,-113.202,171.987,41.121,157.869
C00747=1043.116,298.699,-113.235,171.990,41.123,157.869
C00748=1043.123,298.947,-113.268,171.993,41.126,157.870
C00749=1043.129,299.195,-113.300,171.997,41.128,157.871
C00750=1043.137,299.442,-113.333,172.001,41.131,157.872
C00751=1043.144,299.690,-113.366,172.005,41.133,157.873
C00752=1043.150,299.937,-113.399,172.008,41.136,157.873
C00753=1043.156,300.185,-113.432,172.012,41.138,157.874
C00754=1043.163,300.433,-113.465,172.016,41.141,157.875
C00755=1043.170,300.681,-113.497,172.019,41.143,157.876
C00756=1043.177,300.928,-113.530,172.023,41.145,157.876
C00757=1043.183,301.176,-113.563,172.027,41.148,157.877
C00758=1043.190,301.423,-113.596,172.031,41.151,157.878
C00759=1043.197,301.672,-113.630,172.034,41.153,157.879
C00760=1043.203,301.919,-113.662,172.038,41.156,157.879
C00761=1043.210,302.167,-113.694,172.041,41.158,157.880
C00762=1043.217,302.414,-113.728,172.045,41.161,157.881
C00763=1043.224,302.662,-113.761,172.049,41.163,157.882
C00764=1043.231,302.910,-113.794,172.053,41.166,157.882
C00765=1043.237,303.158,-113.827,172.057,41.169,157.883
C00766=1043.245,303.405,-113.860,172.061,41.171,157.884
C00767=1043.251,303.653,-113.893,172.065,41.173,157.885
C00768=1043.258,303.901,-113.926,172.068,41.176,157.886
C00769=1043.265,304.148,-113.959,172.071,41.179,157.886
C00770=1043.272,304.396,-113.993,172.075,41.181,157.887
C00771=1043.278,304.643,-114.026,172.079,41.184,157.888
C00772=1043.288,304.970,-114.069,172.084,41.187,157.889
C00773=1043.296,305.297,-114.113,172.089,41.191,157.890
C00774=1043.306,305.623,-114.157,172.095,41.194,157.891
C00775=1043.314,305.950,-114.201,172.100,41.197,157.892
C00776=1043.321,306.199,-114.234,172.104,41.200,157.893
C00777=1043.329,306.446,-114.267,172.107,41.202,157.894
C00778=1043.335,306.693,-114.300,172.111,41.205,157.894
C00779=1043.343,306.941,-114.334,172.115,41.207,157.895
C00780=1043.349,307.189,-114.366,172.119,41.210,157.896
C00781=1043.356,307.436,-114.400,172.123,41.213,157.897
C00782=1043.363,307.684,-114.434,172.127,41.215,157.898
C00783=1043.370,307.932,-114.467,172.131,41.218,157.898
C00784=1043.377,308.179,-114.500,172.135,41.220,157.899
C00785=1043.384,308.427,-114.533,172.139,41.223,157.900
C00786=1043.391,308.674,-114.567,172.142,41.226,157.901
C00787=1043.398,308.922,-114.600,172.146,41.228,157.902
C00788=1043.405,309.170,-114.634,172.150,41.231,157.902
C00789=1043.412,309.417,-114.667,172.154,41.233,157.903
C00790=1043.419,309.665,-114.701,172.158,41.236,157.904
C00791=1043.426,309.913,-114.734,172.162,41.239,157.905
C00792=1043.433,310.160,-114.767,172.166,41.241,157.906
C00793=1043.440,310.408,-114.801,172.170,41.244,157.906
C00794=1043.447,310.655,-114.834,172.174,41.246,157.907
C00795=1043.454,310.904,-114.868,172.178,41.249,157.908
C00796=1043.461,311.151,-114.901,172.181,41.252,157.909
C00797=1043.468,311.398,-114.935,172.185,41.254,157.910
C00798=1043.475,311.646,-114.969,172.189,41.257,157.910
C00799=1043.483,311.894,-115.003,172.193,41.259,157.911
C00800=1043.489,312.141,-115.036,172.197,41.262,157.912
C00801=1043.496,312.389,-115.069,172.201,41.265,157.913
C00802=1043.503,312.636,-115.103,172.205,41.268,157.914
C00803=1043.510,312.884,-115.137,172.209,41.270,157.914
C00804=1043.517,313.131,-115.172,172.214,41.273,157.915
C00805=1043.524,313.378,-115.205,172.218,41.276,157.916
C00806=1043.530,313.626,-115.240,172.222,41.279,157.917
C00807=1043.537,313.874,-115.274,172.226,41.281,157.918
C00808=1043.543,314.121,-115.308,172.230,41.284,157.919
C00809=1043.551,314.369,-115.341,172.234,41.287,157.920
C00810=1043.557,314.617,-115.376,172.238,41.290,157.920
C00811=1043.564,314.865,-115.410,172.242,41.293,157.921
C00812=1043.570,315.111,-115.444,172.246,41.295,157.922
C00813=1043.578,315.359,-115.478,172.250,41.299,157.923
C00814=1043.584,315.607,-115.513,172.254,41.301,157.924
C00815=1043.591,315.855,-115.547,172.258,41.304,157.925
C00816=1043.599,316.102,-115.581,172.262,41.307,157.926
C00817=1043.605,316.349,-115.615,172.265,41.310,157.926
C00818=1043.612,316.597,-115.649,172.270,41.313,157.927
C00819=1043.618,316.845,-115.683,172.274,41.315,157.928
C00820=1043.626,317.092,-115.718,172.279,41.318,157.929
C00821=1043.632,317.340,-115.752,172.282,41.321,157.930
C00822=1043.639,317.587,-115.786,172.286,41.324,157.931
C00823=1043.646,317.835,-115.821,172.290,41.327,157.932
C00824=1043.653,318.082,-115.855,172.294,41.329,157.933
C00825=1043.660,318.329,-115.890,172.298,41.333,157.934
C00826=1043.667,318.577,-115.924,172.302,41.335,157.934
C00827=1043.673,318.825,-115.958,172.307,41.338,157.935
C00828=1043.683,319.157,-116.004,172.313,41.342,157.936
C00829=1043.692,319.488,-116.050,172.318,41.346,157.938
C00830=1043.701,319.819,-116.097,172.323,41.350,157.939
C00831=1043.711,320.151,-116.143,172.329,41.354,157.940
C00832=1043.718,320.398,-116.178,172.334,41.356,157.941
C00833=1043.725,320.646,-116.212,172.338,41.360,157.942
C00834=1043.732,320.893,-116.247,172.342,41.362,157.943
C00835=1043.739,321.141,-116.281,172.346,41.365,157.944
C00836=1043.745,321.388,-116.316,172.350,41.368,157.944
C00837=1043.753,321.635,-116.351,172.355,41.371,157.945
C00838=1043.759,321.883,-116.385,172.359,41.374,157.946
C00839=1043.767,322.130,-116.420,172.363,41.377,157.947
C00840=1043.774,322.378,-116.455,172.367,41.380,157.948
C00841=1043.781,322.625,-116.489,172.371,41.383,157.949
C00842=1043.788,322.873,-116.524,172.376,41.386,157.950
C00843=1043.795,323.120,-116.558,172.380,41.389,157.951
C00844=1043.802,323.368,-116.593,172.384,41.392,157.952
C00845=1043.809,323.616,-116.628,172.388,41.395,157.953
C00846=1043.816,323.863,-116.663,172.393,41.398,157.954
C00847=1043.823,324.110,-116.698,172.397,41.401,157.955
C00848=1043.830,324.358,-116.732,172.401,41.403,157.955
C00849=1043.837,324.605,-116.767,172.405,41.406,157.956
C00850=1043.845,324.852,-116.802,172.411,41.409,157.957
C00851=1043.852,325.100,-116.837,172.414,41.412,157.958
C00852=1043.859,325.348,-116.872,172.419,41.415,157.959
C00853=1043.866,325.595,-116.907,172.424,41.418,157.960
C00854=1043.873,325.842,-116.942,172.428,41.421,157.961
C00855=1043.880,326.090,-116.976,172.432,41.424,157.962
C00856=1043.888,326.338,-117.011,172.436,41.427,157.963
C00857=1043.895,326.585,-117.046,172.441,41.430,157.964
C00858=1043.902,326.832,-117.081,172.445,41.433,157.965
C00859=1043.909,327.080,-117.116,172.449,41.436,157.966
C00860=1043.917,327.327,-117.151,172.454,41.439,157.967
C00861=1043.924,327.575,-117.186,172.458,41.442,157.968
C00862=1043.930,327.822,-117.221,172.462,41.445,157.969
C00863=1043.939,328.070,-117.256,172.467,41.448,157.969
C00864=1043.945,328.317,-117.291,172.471,41.451,157.970
C00865=1043.953,328.564,-117.326,172.476,41.455,157.971
C00866=1043.960,328.812,-117.362,172.480,41.457,157.972
C00867=1043.967,329.059,-117.397,172.485,41.460,157.973
C00868=1043.975,329.306,-117.432,172.490,41.463,157.974
C00869=1043.982,329.554,-117.467,172.494,41.466,157.975
C00870=1043.989,329.801,-117.503,172.498,41.469,157.976
C00871=1043.996,330.048,-117.538,172.503,41.473,157.977
C00872=1044.003,330.296,-117.574,172.507,41.476,157.978
C00873=1044.010,330.544,-117.609,172.511,41.479,157.979
C00874=1044.017,330.790,-117.645,172.517,41.482,157.980
C00875=1044.025,331.039,-117.680,172.521,41.486,157.981
C00876=1044.032,331.285,-117.716,172.525,41.489,157.982
C00877=1044.038,331.533,-117.751,172.530,41.492,157.983
C00878=1044.046,331.781,-117.787,172.534,41.495,157.984
C00879=1044.053,332.027,-117.822,172.538,41.499,157.985
C00880=1044.060,332.276,-117.858,172.543,41.502,157.986
C00881=1044.067,332.523,-117.894,172.548,41.505,157.987
C00882=1044.073,332.770,-117.929,172.553,41.508,157.988
C00883=1044.081,333.017,-117.966,172.557,41.511,157.989
C00884=1044.090,333.343,-118.013,172.563,41.516,157.991
C00885=1044.100,333.671,-118.060,172.569,41.520,157.992
C00886=1044.110,333.997,-118.107,172.575,41.524,157.993
C00887=1044.119,334.323,-118.154,172.581,41.528,157.994
C00888=1044.127,334.570,-118.190,172.586,41.532,157.996
C00889=1044.133,334.818,-118.225,172.590,41.535,157.997
C00890=1044.141,335.065,-118.261,172.595,41.538,157.998
C00891=1044.148,335.312,-118.297,172.600,41.541,157.999
C00892=1044.156,335.560,-118.333,172.604,41.545,158.000
C00893=1044.162,335.807,-118.369,172.609,41.548,158.001
C00894=1044.170,336.055,-118.405,172.613,41.551,158.002
C00895=1044.177,336.302,-118.442,172.618,41.554,158.003
C00896=1044.184,336.549,-118.477,172.623,41.558,158.004
C00897=1044.191,336.797,-118.514,172.628,41.561,158.005
C00898=1044.198,337.044,-118.549,172.632,41.565,158.006
C00899=1044.206,337.291,-118.586,172.637,41.568,158.007
C00900=1044.212,337.538,-118.622,172.642,41.571,158.008
C00901=1044.220,337.786,-118.658,172.647,41.574,158.009
C00902=1044.227,338.033,-118.694,172.651,41.578,158.010
C00903=1044.234,338.280,-118.730,172.656,41.581,158.011
C00904=1044.241,338.528,-118.767,172.660,41.585,158.012
C00905=1044.248,338.774,-118.803,172.666,41.588,158.013
C00906=1044.256,339.022,-118.839,172.670,41.592,158.014
C00907=1044.263,339.270,-118.876,172.675,41.595,158.016
C00908=1044.270,339.516,-118.912,172.679,41.598,158.017
C00909=1044.278,339.764,-118.948,172.685,41.602,158.018
C00910=1044.285,340.012,-118.985,172.689,41.606,158.019
C00911=1044.292,340.258,-119.021,172.694,41.609,158.020
C00912=1044.300,340.505,-119.058,172.699,41.612,158.021
C00913=1044.307,340.753,-119.094,172.704,41.616,158.022
C00914=1044.314,341.000,-119.130,172.709,41.619,158.023
C00915=1044.322,341.247,-119.167,172.713,41.623,158.024
C00916=1044.328,341.495,-119.203,172.719,41.626,158.025
C00917=1044.336,341.742,-119.240,172.723,41.629,158.026
C00918=1044.344,341.988,-119.276,172.728,41.633,158.027
C00919=1044.350,342.236,-119.313,172.733,41.636,158.029
C00920=1044.358,342.483,-119.350,172.738,41.640,158.030
C00921=1044.365,342.731,-119.387,172.743,41.644,158.031
C00922=1044.372,342.978,-119.423,172.747,41.647,158.032
C00923=1044.380,343.225,-119.460,172.753,41.651,158.033
C00924=1044.387,343.472,-119.496,172.758,41.654,158.034
C00925=1044.395,343.719,-119.534,172.762,41.658,158.035
C00926=1044.402,343.967,-119.571,172.767,41.661,158.036
C00927=1044.409,344.213,-119.607,172.772,41.665,158.038
C00928=1044.416,344.461,-119.644,172.777,41.668,158.039
C00929=1044.424,344.708,-119.681,172.782,41.672,158.040
C00930=1044.431,344.955,-119.718,172.787,41.676,158.041
C00931=1044.439,345.202,-119.755,172.792,41.679,158.042
C00932=1044.446,345.450,-119.791,172.797,41.683,158.043
C00933=1044.453,345.697,-119.829,172.802,41.686,158.044
C00934=1044.460,345.943,-119.866,172.807,41.690,158.046
C00935=1044.467,346.191,-119.902,172.812,41.693,158.047
C00936=1044.475,346.438,-119.940,172.817,41.698,158.048
C00937=1044.482,346.685,-119.977,172.822,41.701,158.049
C00938=1044.489,346.933,-120.014,172.828,41.705,158.050
C00939=1044.497,347.180,-120.051,172.832,41.709,158.051
C00940=1044.507,347.502,-120.099,172.839,41.713,158.053
C00941=1044.517,347.825,-120.149,172.846,41.718,158.055
C00942=1044.526,348.148,-120.197,172.852,41.723,158.056
C00943=1044.536,348.471,-120.246,172.859,41.728,158.058
C00944=1044.544,348.718,-120.283,172.864,41.732,158.059
C00945=1044.551,348.965,-120.321,172.869,41.735,158.060
C00946=1044.559,349.212,-120.358,172.874,41.739,158.061
C00947=1044.566,349.459,-120.395,172.880,41.743,158.062
C00948=1044.573,349.706,-120.433,172.885,41.746,158.064
C00949=1044.581,349.953,-120.469,172.889,41.750,158.065
C00950=1044.588,350.200,-120.507,172.895,41.754,158.066
C00951=1044.596,350.448,-120.545,172.900,41.758,158.067
C00952=1044.603,350.695,-120.582,172.906,41.761,158.068
C00953=1044.610,350.942,-120.620,172.910,41.766,158.070
C00954=1044.617,351.189,-120.657,172.915,41.769,158.071
C00955=1044.625,351.436,-120.695,172.921,41.773,158.072
C00956=1044.633,351.683,-120.732,172.926,41.777,158.073
C00957=1044.640,351.929,-120.770,172.932,41.781,158.075
C00958=1044.647,352.177,-120.807,172.936,41.784,158.076
C00959=1044.655,352.424,-120.845,172.942,41.789,158.077
C00960=1044.663,352.671,-120.883,172.947,41.792,158.078
C00961=1044.670,352.918,-120.921,172.953,41.796,158.079
C00962=1044.677,353.165,-120.959,172.958,41.800,158.081
C00963=1044.685,353.412,-120.997,172.964,41.804,158.082
C00964=1044.692,353.659,-121.034,172.968,41.808,158.083
C00965=1044.700,353.907,-121.072,172.974,41.812,158.085
C00966=1044.708,354.153,-121.110,172.979,41.816,158.086
C00967=1044.715,354.400,-121.148,172.985,41.820,158.087
C00968=1044.722,354.647,-121.186,172.990,41.824,158.088
C00969=1044.730,354.894,-121.224,172.995,41.827,158.089
C00970=1044.738,355.141,-121.262,173.001,41.832,158.091
C00971=1044.745,355.388,-121.300,173.006,41.836,158.092
C00972=1044.753,355.635,-121.338,173.011,41.840,158.093
C00973=1044.760,355.883,-121.376,173.016,41.843,158.095
C00974=1044.768,356.129,-121.414,173.022,41.847,158.096
C00975=1044.775,356.376,-121.452,173.028,41.852,158.097
C00976=1044.783,356.624,-121.490,173.033,41.856,158.099
C00977=1044.791,356.870,-121.529,173.039,41.860,158.100
C00978=1044.798,357.117,-121.566,173.044,41.864,158.101
C00979=1044.806,357.364,-121.605,173.050,41.868,158.102
C00980=1044.814,357.611,-121.643,173.055,41.872,158.104
C00981=1044.821,357.857,-121.681,173.061,41.876,158.105
C00982=1044.830,358.105,-121.720,173.066,41.880,158.106
C00983=1044.836,358.352,-121.758,173.072,41.884,158.108
C00984=1044.844,358.599,-121.796,173.078,41.888,158.109
C00985=1044.852,358.846,-121.835,173.083,41.892,158.110
C00986=1044.859,359.092,-121.873,173.089,41.896,158.112
C00987=1044.867,359.340,-121.912,173.094,41.901,158.113
C00988=1044.875,359.586,-121.950,173.100,41.905,158.114
C00989=1044.882,359.833,-121.989,173.105,41.909,158.116
C00990=1044.890,360.080,-122.027,173.111,41.913,158.117
C00991=1044.897,360.327,-122.066,173.117,41.917,158.118
C00992=1044.906,360.574,-122.104,173.122,41.921,158.120
C00993=1044.913,360.820,-122.142,173.128,41.926,158.121
C00994=1044.921,361.068,-122.182,173.133,41.930,158.122
C00995=1044.928,361.314,-122.220,173.139,41.934,158.124
C00996=1044.938,361.643,-122.272,173.146,41.939,158.126
C00997=1044.949,361.971,-122.323,173.153,41.946,158.128
C00998=1044.960,362.300,-122.375,173.162,41.951,158.129
C00999=1044.970,362.629,-122.426,173.169,41.957,158.131
C01000=1044.977,362.875,-122.465,173.174,41.961,158.133
C01001=1044.985,363.122,-122.505,173.180,41.965,158.134
C01002=1044.993,363.369,-122.543,173.186,41.970,158.135
C01003=1045.000,363.616,-122.582,173.192,41.974,158.137
C01004=1045.008,363.863,-122.621,173.198,41.978,158.138
C01005=1045.015,364.109,-122.660,173.204,41.983,158.140
C01006=1045.024,364.356,-122.700,173.210,41.987,158.141
C01007=1045.031,364.603,-122.738,173.215,41.991,158.142
C01008=1045.039,364.849,-122.778,173.221,41.996,158.144
C01009=1045.046,365.097,-122.817,173.227,42.000,158.145
C01010=1045.054,365.343,-122.856,173.232,42.005,158.147
C01011=1045.062,365.590,-122.896,173.238,42.009,158.148
C01012=1045.070,365.837,-122.934,173.245,42.014,158.150
C01013=1045.077,366.083,-122.974,173.250,42.018,158.151
C01014=1045.085,366.330,-123.013,173.256,42.022,158.153
C01015=1045.093,366.577,-123.053,173.262,42.027,158.154
C01016=1045.101,366.824,-123.092,173.268,42.032,158.156
C01017=1045.109,367.070,-123.131,173.273,42.036,158.157
C01018=1045.116,367.318,-123.171,173.280,42.040,158.158
C01019=1045.125,367.564,-123.210,173.286,42.045,158.160
C01020=1045.132,367.811,-123.250,173.292,42.049,158.161
C01021=1045.140,368.057,-123.289,173.298,42.054,158.163
C01022=1045.148,368.304,-123.329,173.303,42.059,158.164
C01023=1045.156,368.550,-123.368,173.310,42.063,158.166
C01024=1045.164,368.798,-123.407,173.316,42.068,158.167
C01025=1045.172,369.045,-123.447,173.322,42.072,158.169
C01026=1045.180,369.292,-123.486,173.327,42.077,158.170
C01027=1045.188,369.538,-123.526,173.334,42.081,158.172
C01028=1045.196,369.784,-123.565,173.340,42.086,158.173
C01029=1045.203,370.031,-123.605,173.346,42.091,158.175
C01030=1045.212,370.278,-123.645,173.353,42.095,158.176
C01031=1045.220,370.524,-123.685,173.358,42.100,158.178
C01032=1045.228,370.771,-123.725,173.364,42.104,158.179
C01033=1045.236,371.018,-123.764,173.371,42.109,158.181
C01034=1045.244,371.265,-123.804,173.377,42.114,158.183
C01035=1045.251,371.511,-123.844,173.383,42.118,158.184
C01036=1045.259,371.758,-123.885,173.389,42.123,158.186
C01037=1045.268,372.004,-123.924,173.396,42.128,158.187
C01038=1045.276,372.251,-123.964,173.401,42.133,158.189
C01039=1045.284,372.497,-124.005,173.407,42.137,158.190
C01040=1045.291,372.744,-124.045,173.414,42.142,158.192
C01041=1045.299,372.991,-124.085,173.420,42.147,158.193
C01042=1045.307,373.238,-124.125,173.426,42.152,158.195
C01043=1045.315,373.484,-124.165,173.433,42.156,158.197
C01044=1045.323,373.731,-124.206,173.439,42.162,158.198
C01045=1045.331,373.977,-124.245,173.446,42.166,158.200
C01046=1045.339,374.224,-124.286,173.452,42.171,158.201
C01047=1045.347,374.471,-124.326,173.458,42.176,158.203
C01048=1045.355,374.717,-124.366,173.465,42.181,158.205
C01049=1045.363,374.963,-124.407,173.471,42.186,158.206
C01050=1045.371,375.210,-124.447,173.477,42.190,158.208
C01051=1045.379,375.456,-124.488,173.483,42.195,158.209
C01052=1045.391,375.805,-124.545,173.492,42.203,158.212
C01053=1045.402,376.152,-124.602,173.502,42.209,158.214
C01054=1045.414,376.501,-124.659,173.511,42.216,158.216
C01055=1045.425,376.848,-124.716,173.520,42.223,158.219
C01056=1045.434,377.095,-124.757,173.527,42.228,158.220
C01057=1045.442,377.341,-124.797,173.533,42.233,158.222
C01058=1045.450,377.588,-124.838,173.540,42.238,158.224
C01059=1045.458,377.834,-124.879,173.546,42.243,158.225
C01060=1045.466,378.081,-124.920,173.553,42.248,158.227
C01061=1045.474,378.327,-124.960,173.559,42.253,158.229
C01062=1045.482,378.574,-125.001,173.566,42.258,158.230
C01063=1045.491,378.821,-125.042,173.572,42.263,158.232
C01064=1045.499,379.067,-125.082,173.579,42.269,158.234
C01065=1045.507,379.313,-125.123,173.585,42.274,158.235
C01066=1045.516,379.560,-125.164,173.592,42.279,158.237
C01067=1045.524,379.806,-125.205,173.599,42.284,158.239
C01068=1045.531,380.052,-125.247,173.605,42.289,158.240
C01069=1045.540,380.299,-125.288,173.612,42.294,158.242
C01070=1045.548,380.546,-125.328,173.618,42.299,158.244
C01071=1045.556,380.791,-125.370,173.625,42.304,158.246
C01072=1045.564,381.039,-125.411,173.632,42.310,158.247
C01073=1045.572,381.285,-125.452,173.639,42.315,158.249
C01074=1045.581,381.531,-125.494,173.646,42.320,158.251
C01075=1045.589,381.778,-125.534,173.652,42.326,158.253
C01076=1045.597,382.024,-125.576,173.659,42.331,158.254
C01077=1045.605,382.271,-125.617,173.666,42.336,158.256
C01078=1045.614,382.516,-125.659,173.672,42.341,158.258
C01079=1045.622,382.763,-125.700,173.680,42.347,158.260
C01080=1045.630,383.009,-125.741,173.687,42.352,158.262
C01081=1045.639,383.256,-125.782,173.693,42.357,158.263
C01082=1045.647,383.502,-125.824,173.700,42.363,158.265
C01083=1045.655,383.748,-125.866,173.707,42.368,158.267
C01084=1045.663,383.995,-125.907,173.714,42.373,158.269
C01085=1045.672,384.241,-125.948,173.721,42.379,158.271
C01086=1045.681,384.487,-125.990,173.728,42.384,158.272
C01087=1045.689,384.733,-126.032,173.735,42.389,158.274
C01088=1045.698,384.980,-126.074,173.741,42.395,158.276
C01089=1045.706,385.226,-126.115,173.749,42.400,158.278
C01090=1045.714,385.473,-126.157,173.756,42.406,158.280
C01091=1045.723,385.719,-126.199,173.763,42.411,158.282
C01092=1045.732,385.965,-126.240,173.770,42.417,158.283
C01093=1045.739,386.211,-126.282,173.777,42.423,158.285
C01094=1045.748,386.458,-126.324,173.784,42.428,158.287
C01095=1045.757,386.704,-126.366,173.791,42.434,158.289
C01096=1045.765,386.950,-126.408,173.799,42.439,158.291
C01097=1045.774,387.197,-126.449,173.806,42.444,158.293
C01098=1045.783,387.443,-126.491,173.812,42.450,158.295
C01099=1045.791,387.690,-126.533,173.820,42.456,158.297
C01100=1045.800,387.935,-126.576,173.827,42.461,158.298
C01101=1045.808,388.181,-126.617,173.834,42.467,158.300
C01102=1045.816,388.428,-126.659,173.841,42.472,158.302
C01103=1045.825,388.674,-126.701,173.849,42.478,158.304
C01104=1045.834,388.920,-126.744,173.856,42.483,158.306
C01105=1045.843,389.166,-126.786,173.864,42.489,158.308
C01106=1045.851,389.413,-126.828,173.870,42.495,158.310
C01107=1045.860,389.658,-126.870,173.877,42.501,158.312
C01108=1045.873,390.040,-126.936,173.889,42.510,158.315
C01109=1045.886,390.421,-127.001,173.901,42.518,158.318
C01110=1045.900,390.803,-127.067,173.912,42.528,158.321
C01111=1045.913,391.184,-127.133,173.924,42.537,158.324
C01112=1045.922,391.430,-127.176,173.931,42.543,158.326
C01113=1045.930,391.676,-127.219,173.938,42.548,158.328
C01114=1045.939,391.922,-127.261,173.946,42.554,158.330
C01115=1045.948,392.168,-127.303,173.953,42.560,158.332
C01116=1045.956,392.414,-127.346,173.961,42.566,158.334
C01117=1045.965,392.660,-127.389,173.968,42.572,158.336
C01118=1045.973,392.906,-127.432,173.976,42.577,158.338
C01119=1045.982,393.153,-127.474,173.983,42.583,158.340
C01120=1045.991,393.399,-127.517,173.991,42.589,158.342
C01121=1046.000,393.645,-127.561,173.998,42.595,158.344
C01122=1046.008,393.891,-127.604,174.006,42.601,158.346
C01123=1046.018,394.137,-127.646,174.015,42.608,158.348
C01124=1046.026,394.383,-127.689,174.022,42.614,158.350
C01125=1046.035,394.629,-127.733,174.030,42.620,158.353
C01126=1046.043,394.875,-127.776,174.037,42.626,158.355
C01127=1046.052,395.121,-127.819,174.045,42.632,158.357
C01128=1046.062,395.367,-127.862,174.052,42.638,158.359
C01129=1046.070,395.613,-127.905,174.060,42.644,158.361
C01130=1046.079,395.859,-127.948,174.069,42.650,158.363
C01131=1046.088,396.105,-127.992,174.076,42.656,158.365
C01132=1046.097,396.352,-128.035,174.084,42.662,158.367
C01133=1046.105,396.598,-128.078,174.092,42.668,158.369
C01134=1046.114,396.843,-128.122,174.099,42.675,158.372
C01135=1046.123,397.090,-128.165,174.108,42.681,158.374
C01136=1046.132,397.335,-128.209,174.116,42.687,158.376
C01137=1046.140,397.581,-128.252,174.124,42.694,158.378
C01138=1046.150,397.827,-128.296,174.131,42.700,158.380
C01139=1046.158,398.073,-128.339,174.139,42.706,158.382
C01140=1046.167,398.319,-128.383,174.148,42.713,158.385
C01141=1046.176,398.565,-128.427,174.155,42.718,158.387
C01142=1046.185,398.811,-128.470,174.163,42.725,158.389
C01143=1046.194,399.057,-128.514,174.172,42.731,158.391
C01144=1046.203,399.303,-128.558,174.180,42.738,158.393
C01145=1046.213,399.549,-128.602,174.187,42.744,158.396
C01146=1046.221,399.795,-128.645,174.196,42.751,158.398
C01147=1046.230,400.041,-128.689,174.204,42.757,158.400
C01148=1046.239,400.286,-128.733,174.212,42.764,158.402
C01149=1046.249,400.533,-128.777,174.221,42.770,158.405
C01150=1046.258,400.778,-128.820,174.229,42.776,158.407
C01151=1046.267,401.024,-128.865,174.237,42.783,158.409
C01152=1046.276,401.270,-128.909,174.245,42.789,158.411
C01153=1046.285,401.516,-128.952,174.253,42.796,158.414
C01154=1046.295,401.762,-128.997,174.262,42.803,158.416
C01155=1046.303,402.008,-129.041,174.270,42.809,158.418
C01156=1046.312,402.254,-129.085,174.279,42.816,158.421
C01157=1046.321,402.500,-129.129,174.287,42.822,158.423
C01158=1046.331,402.745,-129.174,174.296,42.829,158.425
C01159=1046.340,402.991,-129.218,174.304,42.836,158.428
C01160=1046.349,403.237,-129.262,174.313,42.842,158.430
C01161=1046.358,403.483,-129.307,174.320,42.849,158.432
C01162=1046.367,403.728,-129.351,174.329,42.856,158.435
C01163=1046.376,403.975,-129.396,174.337,42.862,158.437
C01164=1046.392,404.375,-129.469,174.351,42.874,158.441
C01165=1046.406,404.775,-129.541,174.365,42.884,158.445
C01166=1046.421,405.175,-129.615,174.379,42.896,158.449
C01167=1046.437,405.576,-129.687,174.393,42.907,158.453
C01168=1046.445,405.821,-129.732,174.402,42.914,158.455
C01169=1046.455,406.067,-129.777,174.411,42.921,158.458
C01170=1046.464,406.313,-129.822,174.419,42.928,158.460
C01171=1046.473,406.559,-129.866,174.428,42.935,158.462
C01172=1046.482,406.805,-129.912,174.438,42.941,158.465
C01173=1046.492,407.050,-129.956,174.446,42.949,158.467
C01174=1046.501,407.296,-130.002,174.455,42.956,158.470
C01175=1046.510,407.541,-130.047,174.464,42.962,158.472
C01176=1046.520,407.787,-130.091,174.472,42.970,158.475
C01177=1046.530,408.033,-130.137,174.481,42.977,158.477
C01178=1046.539,408.279,-130.182,174.491,42.984,158.480
C01179=1046.548,408.525,-130.227,174.500,42.991,158.482
C01180=1046.558,408.770,-130.272,174.508,42.998,158.485
C01181=1046.567,409.016,-130.318,174.517,43.005,158.487
C01182=1046.577,409.261,-130.363,174.527,43.012,158.490
C01183=1046.586,409.507,-130.409,174.536,43.019,158.493
C01184=1046.596,409.753,-130.454,174.545,43.027,158.495
C01185=1046.605,409.999,-130.499,174.554,43.034,158.498
C01186=1046.615,410.244,-130.545,174.563,43.041,158.500
C01187=1046.625,410.490,-130.591,174.572,43.049,158.503
C01188=1046.634,410.735,-130.637,174.581,43.056,158.506
C01189=1046.644,410.981,-130.682,174.591,43.063,158.508
C01190=1046.654,411.227,-130.728,174.600,43.070,158.511
C01191=1046.664,411.472,-130.773,174.609,43.077,158.513
C01192=1046.673,411.718,-130.819,174.619,43.085,158.516
C01193=1046.683,411.964,-130.864,174.628,43.092,158.519
C01194=1046.692,412.209,-130.910,174.638,43.100,158.521
C01195=1046.703,412.455,-130.956,174.647,43.107,158.524
C01196=1046.712,412.700,-131.002,174.656,43.114,158.527
C01197=1046.722,412.946,-131.048,174.666,43.122,158.529
C01198=1046.731,413.192,-131.094,174.675,43.129,158.532
C01199=1046.741,413.437,-131.141,174.685,43.137,158.535
C01200=1046.751,413.682,-131.186,174.694,43.144,158.538
C01201=1046.761,413.928,-131.233,174.704,43.152,158.540
C01202=1046.770,414.173,-131.279,174.713,43.160,158.543
C01203=1046.780,414.419,-131.326,174.724,43.167,158.546
C01204=1046.789,414.665,-131.372,174.733,43.175,158.549
C01205=1046.799,414.910,-131.418,174.743,43.183,158.551
C01206=1046.809,415.156,-131.464,174.753,43.191,158.554
C01207=1046.820,415.401,-131.511,174.762,43.198,158.557
C01208=1046.829,415.647,-131.557,174.772,43.206,158.560
C01209=1046.839,415.892,-131.604,174.782,43.214,158.563
C01210=1046.849,416.137,-131.651,174.792,43.222,158.566
C01211=1046.859,416.383,-131.697,174.802,43.229,158.568
C01212=1046.869,416.629,-131.744,174.811,43.237,158.571
C01213=1046.878,416.873,-131.791,174.822,43.245,158.574
C01214=1046.888,417.119,-131.837,174.832,43.252,158.577
C01215=1046.898,417.365,-131.884,174.841,43.261,158.580
C01216=1046.909,417.610,-131.930,174.852,43.268,158.583
C01217=1046.919,417.855,-131.977,174.862,43.276,158.586
C01218=1046.929,418.101,-132.025,174.872,43.284,158.589
C01219=1046.939,418.347,-132.071,174.882,43.292,158.591
C01220=1046.955,418.724,-132.144,174.898,43.304,158.596
C01221=1046.970,419.102,-132.216,174.914,43.317,158.601
C01222=1046.986,419.480,-132.289,174.930,43.330,158.605
C01223=1047.001,419.857,-132.362,174.945,43.342,158.610
C01224=1047.011,420.103,-132.410,174.956,43.350,158.613
C01225=1047.021,420.348,-132.457,174.967,43.358,158.616
C01226=1047.031,420.594,-132.504,174.977,43.367,158.619
C01227=1047.042,420.838,-132.552,174.988,43.375,158.622
C01228=1047.052,421.084,-132.599,174.998,43.383,158.625
C01229=1047.062,421.329,-132.646,175.009,43.391,158.628
C01230=1047.072,421.575,-132.695,175.019,43.400,158.631
C01231=1047.083,421.820,-132.742,175.030,43.408,158.634
C01232=1047.094,422.095,-132.796,175.041,43.418,158.638
C01233=1047.105,422.370,-132.849,175.054,43.426,158.641
C01234=1047.118,422.645,-132.903,175.066,43.436,158.645
C01235=1047.129,422.920,-132.956,175.078,43.446,158.648
C01236=1047.139,423.165,-133.005,175.089,43.454,158.651
C01237=1047.150,423.411,-133.052,175.100,43.462,158.655
C01238=1047.160,423.655,-133.100,175.110,43.471,158.658
C01239=1047.171,423.900,-133.148,175.122,43.480,158.661
C01240=1047.181,424.146,-133.196,175.133,43.488,158.664
C01241=1047.191,424.391,-133.244,175.144,43.497,158.668
C01242=1047.202,424.636,-133.292,175.155,43.505,158.671
C01243=1047.213,424.881,-133.340,175.166,43.514,158.674
C01244=1047.224,425.126,-133.389,175.177,43.522,158.677
C01245=1047.234,425.371,-133.437,175.188,43.531,158.680
C01246=1047.245,425.617,-133.486,175.199,43.540,158.684
C01247=1047.254,425.862,-133.534,175.211,43.549,158.687
C01248=1047.266,426.107,-133.582,175.222,43.557,158.690
C01249=1047.276,426.351,-133.632,175.233,43.566,158.694
C01250=1047.287,426.597,-133.680,175.244,43.575,158.697
C01251=1047.297,426.841,-133.728,175.256,43.584,158.700
C01252=1047.308,427.086,-133.777,175.267,43.593,158.704
C01253=1047.319,427.332,-133.826,175.279,43.602,158.707
C01254=1047.329,427.576,-133.875,175.290,43.610,158.710
C01255=1047.340,427.821,-133.923,175.303,43.619,158.714
C01256=1047.351,428.066,-133.973,175.314,43.628,158.717
C01257=1047.361,428.311,-134.021,175.326,43.637,158.721
C01258=1047.372,428.556,-134.070,175.337,43.646,158.724
C01259=1047.383,428.801,-134.119,175.349,43.656,158.728
C01260=1047.394,429.047,-134.168,175.360,43.665,158.731
C01261=1047.405,429.291,-134.217,175.373,43.673,158.735
C01262=1047.415,429.536,-134.267,175.385,43.683,158.738
C01263=1047.426,429.781,-134.316,175.396,43.692,158.742
C01264=1047.437,430.025,-134.365,175.409,43.701,158.745
C01265=1047.448,430.271,-134.415,175.420,43.710,158.749
C01266=1047.459,430.516,-134.464,175.432,43.720,158.752
C01267=1047.469,430.761,-134.514,175.445,43.729,158.756
C01268=1047.481,431.005,-134.564,175.457,43.738,158.760
C01269=1047.492,431.250,-134.613,175.468,43.748,158.763
C01270=1047.502,431.495,-134.663,175.481,43.757,158.767
C01271=1047.514,431.740,-134.712,175.493,43.766,158.770
C01272=1047.525,431.984,-134.762,175.506,43.776,158.774
C01273=1047.535,432.229,-134.812,175.518,43.786,158.778
C01274=1047.546,432.474,-134.862,175.531,43.795,158.782
C01275=1047.558,432.718,-134.911,175.542,43.804,158.785
C01276=1047.568,432.934,-134.956,175.554,43.813,158.788
C01277=1047.578,433.149,-135.000,175.565,43.821,158.792
C01278=1047.587,433.365,-135.043,175.575,43.830,158.795
C01279=1047.597,433.580,-135.088,175.587,43.838,158.798
C01280=1047.607,433.795,-135.132,175.598,43.846,158.802
C01281=1047.617,434.010,-135.176,175.610,43.855,158.805
C01282=1047.627,434.226,-135.220,175.620,43.864,158.808
C01283=1047.636,434.441,-135.265,175.632,43.872,158.812
C01284=1047.648,434.686,-135.315,175.645,43.882,158.816
C01285=1047.660,434.930,-135.365,175.658,43.891,158.819
C01286=1047.671,435.175,-135.416,175.671,43.901,158.823
C01287=1047.682,435.420,-135.466,175.683,43.911,158.827
C01288=1047.694,435.665,-135.517,175.696,43.921,158.831
C01289=1047.706,435.909,-135.567,175.709,43.931,158.835
C01290=1047.717,436.154,-135.617,175.723,43.941,158.839
C01291=1047.728,436.398,-135.668,175.736,43.951,158.843
C01292=1047.740,436.643,-135.719,175.749,43.961,158.847
C01293=1047.751,436.888,-135.769,175.762,43.970,158.851
C01294=1047.763,437.132,-135.821,175.776,43.981,158.855
C01295=1047.774,437.376,-135.872,175.789,43.991,158.859
C01296=1047.786,437.621,-135.922,175.802,44.001,158.863
C01297=1047.798,437.866,-135.974,175.816,44.011,158.867
C01298=1047.809,438.109,-136.025,175.829,44.021,158.871
C01299=1047.820,438.355,-136.076,175.843,44.032,158.875
C01300=1047.832,438.599,-136.127,175.856,44.042,158.879
C01301=1047.844,438.844,-136.178,175.870,44.052,158.883
C01302=1047.856,439.087,-136.229,175.884,44.062,158.887
C01303=1047.867,439.332,-136.281,175.898,44.073,158.891
C01304=1047.879,439.576,-136.332,175.911,44.083,158.895
C01305=1047.891,439.821,-136.384,175.926,44.093,158.900
C01306=1047.903,440.065,-136.436,175.939,44.103,158.904
C01307=1047.914,440.310,-136.488,175.953,44.114,158.908
C01308=1047.926,440.554,-136.539,175.968,44.124,158.912
C01309=1047.939,440.798,-136.591,175.981,44.135,158.917
C01310=1047.950,441.043,-136.643,175.995,44.146,158.921
C01311=1047.962,441.287,-136.694,176.010,44.156,158.925
C01312=1047.975,441.531,-136.746,176.024,44.167,158.929
C01313=1047.987,441.775,-136.798,176.039,44.178,158.934
C01314=1047.998,442.020,-136.850,176.052,44.188,158.938
C01315=1048.010,442.264,-136.902,176.067,44.199,158.942
C01316=1048.022,442.507,-136.955,176.082,44.209,158.947
C01317=1048.034,442.751,-137.007,176.096,44.221,158.951
C01318=1048.046,442.996,-137.059,176.111,44.231,158.956
C01319=1048.059,443.240,-137.112,176.126,44.242,158.960
C01320=1048.071,443.484,-137.164,176.140,44.253,158.965
C01321=1048.083,443.728,-137.216,176.155,44.264,158.969
C01322=1048.095,443.973,-137.269,176.170,44.275,158.974
C01323=1048.107,444.217,-137.321,176.185,44.285,158.978
C01324=1048.119,444.461,-137.373,176.199,44.297,158.982
C01325=1048.133,444.705,-137.427,176.214,44.308,158.987
C01326=1048.144,444.949,-137.479,176.230,44.319,158.992
C01327=1048.157,445.193,-137.532,176.245,44.330,158.996
C01328=1048.169,445.436,-137.584,176.260,44.341,159.001
C01329=1048.181,445.679,-137.637,176.275,44.352,159.006
C01330=1048.194,445.922,-137.689,176.290,44.363,159.010
C01331=1048.208,446.166,-137.741,176.306,44.374,159.015
C01332=1048.222,446.409,-137.793,176.322,44.385,159.019
C01333=1048.237,446.653,-137.844,176.337,44.395,159.024
C01334=1048.253,446.897,-137.894,176.353,44.406,159.028
C01335=1048.269,447.141,-137.944,176.368,44.416,159.033
C01336=1048.298,447.545,-138.026,176.395,44.433,159.040
C01337=1048.328,447.949,-138.106,176.421,44.450,159.047
C01338=1048.360,448.354,-138.184,176.447,44.466,159.055
C01339=1048.394,448.760,-138.262,176.475,44.481,159.062
C01340=1048.415,449.005,-138.308,176.491,44.491,159.066
C01341=1048.437,449.250,-138.353,176.507,44.500,159.070
C01342=1048.460,449.494,-138.398,176.524,44.509,159.075
C01343=1048.484,449.739,-138.442,176.540,44.518,159.079
C01344=1048.507,449.984,-138.486,176.557,44.527,159.083
C01345=1048.532,450.231,-138.529,176.573,44.535,159.087
C01346=1048.558,450.475,-138.572,176.590,44.544,159.091
C01347=1048.584,450.721,-138.614,176.607,44.552,159.095
C01348=1048.274,450.752,-138.918,176.608,44.641,159.121
C01349=1048.248,450.507,-138.876,176.591,44.633,159.117
C01350=1048.222,450.261,-138.833,176.574,44.624,159.113
C01351=1048.197,450.016,-138.790,176.557,44.616,159.109
C01352=1048.172,449.770,-138.746,176.540,44.607,159.105
C01353=1048.149,449.526,-138.702,176.524,44.598,159.100
C01354=1048.126,449.280,-138.657,176.507,44.590,159.096
C01355=1048.104,449.036,-138.612,176.491,44.580,159.092
C01356=1048.082,448.791,-138.566,176.475,44.571,159.088
C01357=1048.049,448.403,-138.492,176.449,44.556,159.081
C01358=1048.018,448.015,-138.417,176.423,44.541,159.074
C01359=1047.989,447.628,-138.341,176.398,44.525,159.067
C01360=1047.961,447.242,-138.263,176.373,44.509,159.060
C01361=1047.944,446.998,-138.214,176.357,44.500,159.056
C01362=1047.927,446.754,-138.163,176.341,44.489,159.051
C01363=1047.912,446.510,-138.113,176.325,44.478,159.047
C01364=1047.898,446.267,-138.062,176.310,44.468,159.042
C01365=1047.885,446.023,-138.011,176.294,44.457,159.038
C01366=1047.871,445.779,-137.958,176.279,44.446,159.033
C01367=1047.859,445.537,-137.905,176.263,44.435,159.028
C01368=1047.846,445.294,-137.853,176.248,44.424,159.024
C01369=1047.834,445.050,-137.800,176.233,44.413,159.019
C01370=1047.821,444.806,-137.747,176.218,44.402,159.014
C01371=1047.809,444.562,-137.695,176.203,44.391,159.010
C01372=1047.796,444.318,-137.642,176.187,44.380,159.005
C01373=1047.784,444.074,-137.589,176.172,44.369,159.001
C01374=1047.772,443.829,-137.537,176.158,44.358,158.996
C01375=1047.759,443.585,-137.485,176.143,44.347,158.992
C01376=1047.747,443.341,-137.433,176.128,44.336,158.987
C01377=1047.735,443.096,-137.379,176.113,44.326,158.983
C01378=1047.723,442.853,-137.327,176.099,44.315,158.978
C01379=1047.711,442.609,-137.275,176.084,44.304,158.974
C01380=1047.699,442.365,-137.223,176.069,44.294,158.970
C01381=1047.687,442.121,-137.170,176.055,44.283,158.965
C01382=1047.674,441.876,-137.118,176.040,44.272,158.961
C01383=1047.662,441.632,-137.066,176.025,44.262,158.957
C01384=1047.650,441.388,-137.014,176.012,44.251,158.952
C01385=1047.638,441.144,-136.962,175.997,44.241,158.948
C01386=1047.626,440.899,-136.911,175.983,44.230,158.944
C01387=1047.614,440.655,-136.859,175.968,44.220,158.939
C01388=1047.603,440.410,-136.807,175.955,44.209,158.935
C01389=1047.591,440.166,-136.755,175.941,44.199,158.931
C01390=1047.579,439.922,-136.703,175.926,44.189,158.927
C01391=1047.567,439.678,-136.652,175.913,44.178,158.922
C01392=1047.556,439.434,-136.601,175.899,44.168,158.918
C01393=1047.544,439.189,-136.549,175.884,44.158,158.914
C01394=1047.532,438.945,-136.498,175.871,44.147,158.910
C01395=1047.520,438.700,-136.447,175.857,44.137,158.906
C01396=1047.508,438.456,-136.395,175.844,44.127,158.902
C01397=1047.497,438.212,-136.344,175.829,44.117,158.898
C01398=1047.485,437.967,-136.293,175.816,44.107,158.894
C01399=1047.473,437.722,-136.242,175.802,44.097,158.890
C01400=1047.461,437.478,-136.191,175.789,44.087,158.885
C01401=1047.450,437.234,-136.140,175.776,44.076,158.881
C01402=1047.439,436.989,-136.089,175.762,44.067,158.878
C01403=1047.427,436.745,-136.038,175.749,44.057,158.873
C01404=1047.416,436.500,-135.987,175.736,44.047,158.870
C01405=1047.404,436.255,-135.936,175.722,44.037,158.866
C01406=1047.393,436.011,-135.885,175.709,44.027,158.862
C01407=1047.381,435.766,-135.835,175.696,44.017,158.858
C01408=1047.370,435.522,-135.785,175.683,44.008,158.854
C01409=1047.358,435.277,-135.734,175.670,43.998,158.850
C01410=1047.347,435.033,-135.683,175.657,43.988,158.846
C01411=1047.335,434.788,-135.633,175.644,43.978,158.842
C01412=1047.323,434.544,-135.583,175.631,43.969,158.838
C01413=1047.314,434.327,-135.538,175.620,43.960,158.835
C01414=1047.303,434.110,-135.494,175.608,43.951,158.832
C01415=1047.293,433.894,-135.450,175.597,43.943,158.828
C01416=1047.284,433.678,-135.405,175.585,43.935,158.825
C01417=1047.274,433.462,-135.361,175.575,43.926,158.822
C01418=1047.264,433.245,-135.317,175.564,43.918,158.818
C01419=1047.254,433.028,-135.272,175.552,43.910,158.815
C01420=1047.244,432.812,-135.228,175.541,43.901,158.812
C01421=1047.233,432.567,-135.178,175.529,43.891,158.808
C01422=1047.222,432.323,-135.129,175.516,43.882,158.804
C01423=1047.211,432.078,-135.079,175.504,43.873,158.801
C01424=1047.200,431.834,-135.029,175.491,43.863,158.797
C01425=1047.189,431.589,-134.980,175.479,43.854,158.793
C01426=1047.178,431.344,-134.929,175.466,43.845,158.790
C01427=1047.167,431.099,-134.880,175.455,43.835,158.786
C01428=1047.156,430.854,-134.830,175.442,43.826,158.783
C01429=1047.145,430.610,-134.781,175.430,43.817,158.779
C01430=1047.134,430.365,-134.731,175.417,43.808,158.775
C01431=1047.123,430.120,-134.681,175.406,43.799,158.772
C01432=1047.112,429.875,-134.632,175.394,43.789,158.768
C01433=1047.101,429.630,-134.583,175.381,43.780,158.765
C01434=1047.090,429.385,-134.533,175.370,43.771,158.761
C01435=1047.079,429.140,-134.484,175.358,43.762,158.758
C01436=1047.069,428.895,-134.435,175.347,43.753,158.754
C01437=1047.059,428.650,-134.386,175.334,43.744,158.751
C01438=1047.047,428.406,-134.337,175.322,43.735,158.747
C01439=1047.036,428.161,-134.288,175.311,43.726,158.744
C01440=1047.025,427.915,-134.239,175.299,43.717,158.740
C01441=1047.015,427.671,-134.190,175.288,43.708,158.737
C01442=1047.004,427.426,-134.141,175.275,43.699,158.733
C01443=1046.993,427.181,-134.092,175.264,43.690,158.730
C01444=1046.982,426.935,-134.043,175.253,43.682,158.727
C01445=1046.972,426.691,-133.995,175.241,43.673,158.723
C01446=1046.961,426.445,-133.946,175.230,43.664,158.720
C01447=1046.951,426.201,-133.898,175.218,43.655,158.717
C01448=1046.940,425.955,-133.850,175.207,43.647,158.713
C01449=1046.930,425.711,-133.800,175.195,43.638,158.710
C01450=1046.919,425.466,-133.752,175.184,43.629,158.707
C01451=1046.909,425.221,-133.704,175.173,43.621,158.703
C01452=1046.898,424.975,-133.655,175.162,43.612,158.700
C01453=1046.887,424.731,-133.607,175.150,43.604,158.697
C01454=1046.877,424.485,-133.558,175.139,43.595,158.694
C01455=1046.866,424.240,-133.510,175.128,43.587,158.690
C01456=1046.856,423.994,-133.463,175.118,43.578,158.687
C01457=1046.845,423.750,-133.415,175.106,43.569,158.684
C01458=1046.835,423.504,-133.366,175.095,43.561,158.681
C01459=1046.824,423.259,-133.318,175.084,43.553,158.678
C01460=1046.814,423.014,-133.271,175.073,43.544,158.674
C01461=1046.803,422.769,-133.223,175.063,43.536,158.671
C01462=1046.793,422.523,-133.175,175.052,43.527,158.668
C01463=1046.782,422.279,-133.128,175.041,43.519,158.665
C01464=1046.772,422.033,-133.079,175.030,43.511,158.662
C01465=1046.762,421.788,-133.031,175.020,43.503,158.659
C01466=1046.751,421.543,-132.984,175.008,43.494,158.656
C01467=1046.741,421.298,-132.936,174.997,43.486,158.653
C01468=1046.731,421.053,-132.889,174.988,43.478,158.649
C01469=1046.721,420.807,-132.841,174.977,43.470,158.646
C01470=1046.711,420.562,-132.794,174.967,43.461,158.643
C01471=1046.700,420.316,-132.746,174.956,43.453,158.640
C01472=1046.690,420.071,-132.699,174.946,43.445,158.637
C01473=1046.673,419.662,-132.619,174.928,43.432,158.632
C01474=1046.657,419.252,-132.541,174.911,43.418,158.627
C01475=1046.640,418.843,-132.462,174.893,43.405,158.622
C01476=1046.623,418.433,-132.383,174.876,43.391,158.617
C01477=1046.612,418.187,-132.336,174.866,43.384,158.614
C01478=1046.602,417.941,-132.290,174.855,43.376,158.611
C01479=1046.592,417.696,-132.243,174.845,43.368,158.609
C01480=1046.582,417.451,-132.195,174.836,43.360,158.606
C01481=1046.572,417.205,-132.149,174.825,43.352,158.603
C01482=1046.563,416.960,-132.102,174.815,43.344,158.600
C01483=1046.553,416.715,-132.055,174.806,43.336,158.597
C01484=1046.543,416.469,-132.008,174.795,43.329,158.594
C01485=1046.532,416.224,-131.962,174.785,43.321,158.591
C01486=1046.522,415.978,-131.915,174.776,43.313,158.589
C01487=1046.512,415.733,-131.869,174.765,43.306,158.586
C01488=1046.503,415.487,-131.822,174.755,43.298,158.583
C01489=1046.493,415.241,-131.776,174.746,43.290,158.580
C01490=1046.483,414.997,-131.729,174.736,43.282,158.577
C01491=1046.473,414.751,-131.683,174.726,43.275,158.574
C01492=1046.463,414.505,-131.637,174.716,43.268,158.572
C01493=1046.447,414.099,-131.559,174.700,43.255,158.567
C01494=1046.431,413.691,-131.483,174.684,43.242,158.562
C01495=1046.415,413.284,-131.407,174.668,43.230,158.558
C01496=1046.399,412.878,-131.330,174.652,43.218,158.553
C01497=1046.389,412.631,-131.284,174.643,43.210,158.551
C01498=1046.380,412.386,-131.238,174.633,43.202,158.548
C01499=1046.369,412.141,-131.192,174.624,43.195,158.545
C01500=1046.360,411.894,-131.146,174.615,43.188,158.543
C01501=1046.350,411.649,-131.100,174.605,43.181,158.540
C01502=1046.340,411.404,-131.055,174.596,43.173,158.537
C01503=1046.331,411.157,-131.009,174.586,43.166,158.535
C01504=1046.321,410.913,-130.963,174.577,43.159,158.532
C01505=1046.311,410.666,-130.918,174.568,43.151,158.530
C01506=1046.301,410.421,-130.872,174.558,43.144,158.527
C01507=1046.292,410.175,-130.827,174.549,43.137,158.524
C01508=1046.282,409.930,-130.782,174.540,43.130,158.522
C01509=1046.273,409.684,-130.735,174.530,43.123,158.519
C01510=1046.263,409.438,-130.690,174.521,43.116,158.517
C01511=1046.254,409.193,-130.645,174.513,43.109,158.514
C01512=1046.244,408.947,-130.600,174.504,43.101,158.511
C01513=1046.234,408.701,-130.554,174.494,43.095,158.509
C01514=1046.225,408.456,-130.509,174.485,43.087,158.506
C01515=1046.216,408.210,-130.463,174.476,43.080,158.504
C01516=1046.206,407.964,-130.419,174.467,43.074,158.501
C01517=1046.197,407.719,-130.373,174.458,43.066,158.499
C01518=1046.187,407.473,-130.328,174.449,43.059,158.496
C01519=1046.178,407.227,-130.283,174.440,43.053,158.494
C01520=1046.168,406.982,-130.238,174.431,43.046,158.491
C01521=1046.159,406.736,-130.193,174.423,43.038,158.489
C01522=1046.150,406.490,-130.148,174.414,43.031,158.486
C01523=1046.140,406.245,-130.103,174.405,43.025,158.484
C01524=1046.131,405.998,-130.058,174.396,43.018,158.481
C01525=1046.122,405.755,-130.014,174.387,43.011,158.479
C01526=1046.113,405.512,-129.969,174.379,43.004,158.477
C01527=1046.103,405.269,-129.925,174.370,42.998,158.474
C01528=1046.095,405.025,-129.880,174.361,42.991,158.472
C01529=1046.086,404.783,-129.837,174.353,42.984,158.469
C01530=1046.076,404.540,-129.792,174.344,42.978,158.467
C01531=1046.067,404.296,-129.748,174.336,42.971,158.465
C01532=1046.058,404.053,-129.703,174.327,42.964,158.462
C01533=1046.049,403.808,-129.660,174.319,42.957,158.460
C01534=1046.040,403.561,-129.615,174.310,42.951,158.458
C01535=1046.030,403.316,-129.570,174.302,42.944,158.455
C01536=1046.021,403.069,-129.526,174.293,42.937,158.453
C01537=1046.012,402.823,-129.481,174.285,42.931,158.451
C01538=1046.003,402.578,-129.437,174.276,42.924,158.448
C01539=1045.994,402.332,-129.393,174.268,42.918,158.446
C01540=1045.984,402.086,-129.349,174.260,42.911,158.444
C01541=1045.976,401.840,-129.305,174.252,42.904,158.441
C01542=1045.967,401.594,-129.260,174.243,42.898,158.439
C01543=1045.958,401.348,-129.216,174.235,42.891,158.437
C01544=1045.948,401.103,-129.172,174.226,42.885,158.434
C01545=1045.939,400.857,-129.127,174.218,42.879,158.432
C01546=1045.930,400.612,-129.084,174.210,42.872,158.430
C01547=1045.921,400.365,-129.040,174.201,42.865,158.428
C01548=1045.912,400.119,-128.996,174.193,42.859,158.425
C01549=1045.903,399.873,-128.952,174.185,42.853,158.423
C01550=1045.893,399.627,-128.908,174.177,42.847,158.421
C01551=1045.885,399.382,-128.865,174.169,42.840,158.419
C01552=1045.875,399.136,-128.820,174.160,42.834,158.416
C01553=1045.867,398.889,-128.777,174.153,42.827,158.414
C01554=1045.857,398.643,-128.733,174.145,42.821,158.412
C01555=1045.849,398.398,-128.690,174.136,42.815,158.410
C01556=1045.839,398.151,-128.646,174.128,42.809,158.408
C01557=1045.831,397.906,-128.602,174.120,42.802,158.405
C01558=1045.822,397.660,-128.559,174.113,42.796,158.403
C01559=1045.813,397.414,-128.515,174.104,42.790,158.401
C01560=1045.804,397.168,-128.472,174.096,42.784,158.399
C01561=1045.795,396.922,-128.429,174.089,42.777,158.397
C01562=1045.786,396.675,-128.385,174.081,42.771,158.395
C01563=1045.778,396.430,-128.341,174.072,42.765,158.392
C01564=1045.769,396.184,-128.298,174.065,42.759,158.390
C01565=1045.760,395.938,-128.255,174.057,42.753,158.388
C01566=1045.751,395.692,-128.211,174.049,42.747,158.386
C01567=1045.742,395.446,-128.169,174.042,42.741,158.384
C01568=1045.733,395.200,-128.126,174.033,42.735,158.382
C01569=1045.724,394.954,-128.082,174.026,42.729,158.380
C01570=1045.715,394.708,-128.039,174.018,42.722,158.378
C01571=1045.707,394.462,-127.996,174.010,42.716,158.376
C01572=1045.698,394.216,-127.953,174.003,42.710,158.374
C01573=1045.689,393.970,-127.910,173.995,42.705,158.371
C01574=1045.681,393.724,-127.867,173.987,42.699,158.369
C01575=1045.672,393.478,-127.824,173.979,42.693,158.367
C01576=1045.663,393.232,-127.782,173.971,42.687,158.365
C01577=1045.654,392.985,-127.738,173.964,42.681,158.363
C01578=1045.645,392.739,-127.695,173.956,42.675,158.361
C01579=1045.637,392.493,-127.652,173.949,42.669,158.359
C01580=1045.628,392.247,-127.610,173.941,42.663,158.357
C01581=1045.619,392.001,-127.568,173.934,42.657,158.355
C01582=1045.611,391.755,-127.524,173.926,42.651,158.353
C01583=1045.602,391.509,-127.482,173.919,42.646,158.351
C01584=1045.593,391.263,-127.439,173.911,42.640,158.349
C01585=1045.580,390.879,-127.374,173.899,42.631,158.346
C01586=1045.567,390.496,-127.307,173.888,42.622,158.343
C01587=1045.553,390.113,-127.241,173.877,42.613,158.340
C01588=1045.540,389.729,-127.175,173.865,42.604,158.337
C01589=1045.531,389.484,-127.133,173.858,42.599,158.335
C01590=1045.523,389.237,-127.090,173.850,42.593,158.333
C01591=1045.514,388.991,-127.049,173.843,42.587,158.331
C01592=1045.505,388.745,-127.006,173.835,42.582,158.329
C01593=1045.496,388.498,-126.964,173.828,42.576,158.327
C01594=1045.489,388.252,-126.922,173.821,42.571,158.325
C01595=1045.479,388.006,-126.879,173.814,42.565,158.323
C01596=1045.471,387.760,-126.838,173.807,42.559,158.321
C01597=1045.462,387.513,-126.795,173.800,42.554,158.320
C01598=1045.453,387.267,-126.754,173.792,42.548,158.318
C01599=1045.444,387.021,-126.712,173.785,42.543,158.316
C01600=1045.437,386.775,-126.670,173.778,42.537,158.314
C01601=1045.428,386.528,-126.628,173.770,42.532,158.312
C01602=1045.419,386.282,-126.587,173.763,42.526,158.310
C01603=1045.411,386.035,-126.544,173.757,42.521,158.309
C01604=1045.403,385.790,-126.503,173.750,42.516,158.307
C01605=1045.394,385.543,-126.461,173.742,42.510,158.305
C01606=1045.385,385.297,-126.419,173.735,42.505,158.303
C01607=1045.377,385.051,-126.378,173.728,42.499,158.301
C01608=1045.368,384.805,-126.336,173.722,42.494,158.299
C01609=1045.360,384.558,-126.294,173.714,42.489,158.297
C01610=1045.352,384.312,-126.253,173.707,42.483,158.296
C01611=1045.343,384.065,-126.211,173.700,42.478,158.294
C01612=1045.335,383.820,-126.170,173.694,42.473,158.292
C01613=1045.327,383.572,-126.128,173.686,42.467,158.290
C01614=1045.318,383.326,-126.087,173.679,42.462,158.288
C01615=1045.309,383.080,-126.045,173.672,42.457,158.287
C01616=1045.302,382.833,-126.004,173.666,42.451,158.285
C01617=1045.293,382.587,-125.962,173.659,42.446,158.283
C01618=1045.284,382.341,-125.921,173.652,42.441,158.281
C01619=1045.276,382.095,-125.880,173.645,42.436,158.279
C01620=1045.269,381.849,-125.838,173.638,42.431,158.278
C01621=1045.260,381.602,-125.797,173.631,42.425,158.276
C01622=1045.252,381.356,-125.756,173.625,42.420,158.274
C01623=1045.243,381.109,-125.715,173.618,42.415,158.272
C01624=1045.236,380.862,-125.673,173.612,42.410,158.271
C01625=1045.227,380.616,-125.632,173.604,42.405,158.269
C01626=1045.219,380.370,-125.591,173.597,42.400,158.267
C01627=1045.211,380.124,-125.550,173.591,42.394,158.265
C01628=1045.203,379.877,-125.508,173.584,42.389,158.264
C01629=1045.195,379.631,-125.467,173.578,42.384,158.262
C01630=1045.187,379.384,-125.427,173.571,42.379,158.260
C01631=1045.178,379.137,-125.386,173.564,42.374,158.259
C01632=1045.170,378.891,-125.345,173.558,42.369,158.257
C01633=1045.162,378.645,-125.305,173.551,42.364,158.255
C01634=1045.153,378.398,-125.263,173.545,42.359,158.254
C01635=1045.145,378.152,-125.222,173.538,42.354,158.252
C01636=1045.137,377.906,-125.182,173.532,42.349,158.250
C01637=1045.129,377.658,-125.141,173.524,42.344,158.248
C01638=1045.121,377.412,-125.101,173.518,42.339,158.247
C01639=1045.113,377.166,-125.060,173.512,42.334,158.245
C01640=1045.105,376.919,-125.019,173.506,42.329,158.244
C01641=1045.093,376.569,-124.962,173.496,42.322,158.241
C01642=1045.081,376.219,-124.904,173.487,42.315,158.239
C01643=1045.069,375.870,-124.846,173.477,42.308,158.237
C01644=1045.057,375.520,-124.789,173.468,42.301,158.234
C01645=1045.050,375.273,-124.749,173.462,42.296,158.233
C01646=1045.042,375.026,-124.708,173.455,42.291,158.231
C01647=1045.033,374.780,-124.668,173.449,42.287,158.229
C01648=1045.026,374.533,-124.628,173.442,42.282,158.228
C01649=1045.018,374.287,-124.587,173.436,42.277,158.226
C01650=1045.010,374.040,-124.547,173.429,42.272,158.225
C01651=1045.001,373.794,-124.507,173.424,42.268,158.223
C01652=1044.993,373.548,-124.467,173.418,42.263,158.221
C01653=1044.986,373.301,-124.427,173.411,42.258,158.220
C01654=1044.978,373.054,-124.387,173.405,42.253,158.218
C01655=1044.970,372.808,-124.346,173.399,42.248,158.217
C01656=1044.962,372.561,-124.306,173.392,42.244,158.215
C01657=1044.954,372.315,-124.266,173.386,42.239,158.213
C01658=1044.946,372.068,-124.226,173.379,42.234,158.212
C01659=1044.938,371.821,-124.186,173.373,42.230,158.210
C01660=1044.930,371.575,-124.146,173.367,42.225,158.209
C01661=1044.922,371.328,-124.106,173.361,42.220,158.207
C01662=1044.914,371.081,-124.066,173.355,42.216,158.206
C01663=1044.906,370.835,-124.025,173.349,42.211,158.204
C01664=1044.898,370.588,-123.986,173.343,42.206,158.203
C01665=1044.890,370.341,-123.946,173.336,42.202,158.201
C01666=1044.882,370.095,-123.907,173.330,42.197,158.200
C01667=1044.874,369.848,-123.867,173.324,42.192,158.198
C01668=1044.866,369.601,-123.827,173.318,42.188,158.197
C01669=1044.858,369.354,-123.788,173.312,42.184,158.195
C01670=1044.850,369.107,-123.748,173.306,42.179,158.194
C01671=1044.842,368.861,-123.709,173.299,42.175,158.192
C01672=1044.835,368.614,-123.669,173.293,42.170,158.191
C01673=1044.826,368.368,-123.629,173.288,42.166,158.189
C01674=1044.818,368.121,-123.590,173.282,42.161,158.188
C01675=1044.810,367.874,-123.551,173.275,42.156,158.186
C01676=1044.802,367.627,-123.511,173.269,42.152,158.185
C01677=1044.795,367.381,-123.472,173.264,42.148,158.183
C01678=1044.787,367.134,-123.432,173.258,42.143,158.182
C01679=1044.778,366.887,-123.393,173.252,42.139,158.180
C01680=1044.771,366.640,-123.354,173.245,42.134,158.179
C01681=1044.764,366.394,-123.314,173.240,42.130,158.177
C01682=1044.755,366.147,-123.275,173.234,42.126,158.176
C01683=1044.748,365.900,-123.236,173.228,42.121,158.174
C01684=1044.740,365.653,-123.196,173.222,42.116,158.173
C01685=1044.732,365.407,-123.157,173.217,42.112,158.172
C01686=1044.724,365.160,-123.118,173.210,42.108,158.170
C01687=1044.717,364.913,-123.078,173.204,42.104,158.169
C01688=1044.709,364.666,-123.040,173.198,42.099,158.167
C01689=1044.701,364.419,-123.000,173.193,42.094,158.166
C01690=1044.694,364.173,-122.962,173.187,42.090,158.164
C01691=1044.686,363.926,-122.922,173.181,42.086,158.163
C01692=1044.678,363.679,-122.883,173.176,42.082,158.162
C01693=1044.671,363.432,-122.844,173.170,42.077,158.160
C01694=1044.663,363.185,-122.805,173.163,42.073,158.159
C01695=1044.656,362.939,-122.765,173.158,42.069,158.157
C01696=1044.647,362.692,-122.727,173.152,42.065,158.156
C01697=1044.638,362.362,-122.675,173.145,42.059,158.154
C01698=1044.626,362.031,-122.623,173.136,42.053,158.152
C01699=1044.617,361.701,-122.571,173.129,42.048,158.150
C01700=1044.606,361.370,-122.519,173.121,42.042,158.149
C01701=1044.598,361.123,-122.481,173.115,42.038,158.147
C01702=1044.591,360.876,-122.442,173.110,42.034,158.146
C01703=1044.583,360.629,-122.404,173.104,42.030,158.144
C01704=1044.575,360.382,-122.365,173.099,42.025,158.143
C01705=1044.567,360.136,-122.327,173.093,42.021,158.142
C01706=1044.560,359.888,-122.287,173.087,42.017,158.140
C01707=1044.552,359.642,-122.249,173.082,42.013,158.139
C01708=1044.544,359.394,-122.211,173.076,42.009,158.138
C01709=1044.537,359.148,-122.172,173.071,42.005,158.137
C01710=1044.529,358.901,-122.134,173.065,42.001,158.135
C01711=1044.521,358.654,-122.096,173.059,41.997,158.134
C01712=1044.514,358.407,-122.057,173.054,41.993,158.133
C01713=1044.506,358.160,-122.018,173.048,41.989,158.131
C01714=1044.498,357.914,-121.980,173.043,41.985,158.130
C01715=1044.491,357.667,-121.942,173.037,41.981,158.129
C01716=1044.483,357.419,-121.904,173.032,41.977,158.127
C01717=1044.476,357.173,-121.865,173.026,41.973,158.126
C01718=1044.468,356.926,-121.827,173.020,41.968,158.125
C01719=1044.461,356.678,-121.789,173.016,41.964,158.123
C01720=1044.453,356.432,-121.751,173.010,41.960,158.122
C01721=1044.445,356.185,-121.713,173.005,41.957,158.121
C01722=1044.437,355.938,-121.675,172.999,41.953,158.119
C01723=1044.430,355.691,-121.637,172.994,41.948,158.118
C01724=1044.422,355.445,-121.598,172.988,41.944,158.117
C01725=1044.414,355.197,-121.561,172.983,41.941,158.116
C01726=1044.407,354.950,-121.522,172.977,41.937,158.114
C01727=1044.399,354.703,-121.485,172.972,41.933,158.113
C01728=1044.392,354.457,-121.447,172.966,41.929,158.112
C01729=1044.384,354.209,-121.409,172.961,41.925,158.110
C01730=1044.377,353.962,-121.371,172.955,41.921,158.109
C01731=1044.369,353.715,-121.333,172.951,41.917,158.108
C01732=1044.362,353.468,-121.295,172.945,41.913,158.107
C01733=1044.354,353.221,-121.257,172.940,41.910,158.106
C01734=1044.347,352.974,-121.219,172.934,41.906,158.104
C01735=1044.339,352.726,-121.182,172.929,41.902,158.103
C01736=1044.332,352.480,-121.143,172.923,41.898,158.102
C01737=1044.325,352.233,-121.106,172.919,41.894,158.101
C01738=1044.317,351.986,-121.068,172.913,41.890,158.099
C01739=1044.310,351.738,-121.031,172.908,41.887,158.098
C01740=1044.303,351.492,-120.993,172.903,41.883,158.097
C01741=1044.295,351.245,-120.956,172.897,41.879,158.096
C01742=1044.287,350.997,-120.918,172.893,41.875,158.094
C01743=1044.279,350.750,-120.880,172.887,41.871,158.093
C01744=1044.272,350.503,-120.843,172.882,41.868,158.092
C01745=1044.265,350.256,-120.805,172.876,41.864,158.091
C01746=1044.258,350.009,-120.768,172.871,41.860,158.090
C01747=1044.250,349.762,-120.731,172.867,41.857,158.088
C01748=1044.243,349.515,-120.693,172.861,41.852,158.087
C01749=1044.235,349.268,-120.656,172.856,41.849,158.086
C01750=1044.228,349.021,-120.618,172.850,41.845,158.085
C01751=1044.220,348.774,-120.581,172.845,41.842,158.084
C01752=1044.213,348.527,-120.544,172.841,41.838,158.082
C01753=1044.203,348.202,-120.495,172.834,41.833,158.081
C01754=1044.193,347.877,-120.445,172.827,41.828,158.079
C01755=1044.183,347.552,-120.397,172.820,41.823,158.078
C01756=1044.173,347.228,-120.348,172.813,41.819,158.076
C01757=1044.166,346.981,-120.311,172.808,41.815,158.075
C01758=1044.159,346.733,-120.273,172.804,41.811,158.074
C01759=1044.151,346.487,-120.237,172.798,41.808,158.073
C01760=1044.144,346.239,-120.200,172.793,41.804,158.072
C01761=1044.137,345.992,-120.162,172.789,41.801,158.070
C01762=1044.129,345.745,-120.126,172.783,41.797,158.069
C01763=1044.122,345.498,-120.089,172.778,41.794,158.068
C01764=1044.115,345.251,-120.051,172.774,41.790,158.067
C01765=1044.107,345.003,-120.015,172.768,41.786,158.066
C01766=1044.100,344.756,-119.977,172.763,41.783,158.065
C01767=1044.092,344.509,-119.941,172.758,41.779,158.064
C01768=1044.086,344.262,-119.904,172.753,41.776,158.062
C01769=1044.078,344.015,-119.867,172.748,41.772,158.061
C01770=1044.071,343.768,-119.830,172.743,41.768,158.060
C01771=1044.064,343.520,-119.793,172.738,41.765,158.059
C01772=1044.056,343.273,-119.756,172.733,41.761,158.058
C01773=1044.049,343.026,-119.720,172.729,41.758,158.057
C01774=1044.041,342.779,-119.683,172.723,41.755,158.056
C01775=1044.035,342.531,-119.646,172.719,41.751,158.054
C01776=1044.027,342.285,-119.609,172.714,41.747,158.053
C01777=1044.020,342.038,-119.573,172.708,41.744,158.052
C01778=1044.013,341.790,-119.537,172.704,41.741,158.051
C01779=1044.006,341.542,-119.500,172.699,41.737,158.050
C01780=1043.998,341.295,-119.463,172.694,41.733,158.049
C01781=1043.990,341.048,-119.427,172.689,41.730,158.048
C01782=1043.984,340.801,-119.390,172.684,41.727,158.047
